// TIA Portal V15.1 export
// export: Created 2024-06-21T08:41:00.9803831Z, ExportSetting WithDefaults, DisplayName Totally Integrated Automation Portal, DisplayVersion V15.1 Update 5, DisplayName TIA Portal Openness, DisplayVersion V15.1 Update 5, DisplayName SINAMICS Startdrive Advanced, DisplayVersion V15.1, DisplayName G130, G150, S120, S150, SINAMICS MV, S210, DisplayVersion V15.1, DisplayName G110M, G120, G120C, G120D, G120P, DisplayVersion V15.1, DisplayName STEP 7 Professional, DisplayVersion V15.1 Update 5, DisplayName STEP 7 Safety, DisplayVersion V15.1, DisplayName WinCC Professional, DisplayVersion V15.1 Update 5, DisplayName SIMATIC Visualization Architect, DisplayVersion V15.1
FUNCTION_BLOCK "LMode"   // FB1000, FBD
TITLE = LMode
{ S7_Optimized_Access := 'FALSE' }
AUTHOR : VCC
FAMILY : Control
NAME : Mode
VERSION : 1.0
// ================================================================================
// This module is used to handle all operating modes for a modezone as well as 
// resetting of alarms. It get the input from LModeSelector.
// ================================================================================
// stored: AutoNumber false, IsIECCheckEnabled false, SetENOAutomatically False, UDAEnableTagReadback false
   VAR_INPUT
      I_NormalStop { ExternalAccessible := 'False'; ExternalVisible := 'False'; ExternalWritable := 'False'} : Bool;   // Normal Stop Activated Stop Automatic
      I_EnableAlarms { ExternalAccessible := 'False'; ExternalVisible := 'False'; ExternalWritable := 'False'} : Bool;   // Filter alarms for lower levels
      I_AutoModeSel { ExternalAccessible := 'False'; ExternalVisible := 'False'; ExternalWritable := 'False'} : Bool;   // Auto selected
      I_StepModeSel { ExternalAccessible := 'False'; ExternalVisible := 'False'; ExternalWritable := 'False'} : Bool;   // Step selected
      I_HomeRunModeSel { ExternalAccessible := 'False'; ExternalVisible := 'False'; ExternalWritable := 'False'} : Bool;   // Homerun selected
      I_HomeRunPush { ExternalAccessible := 'False'; ExternalVisible := 'False'; ExternalWritable := 'False'} : Bool;   // The reset button needs to be active during the homerun
      I_ManualModeSel { ExternalAccessible := 'False'; ExternalVisible := 'False'; ExternalWritable := 'False'} : Bool;   // Manual selected
      I_ForcedManActSel { ExternalAccessible := 'False'; ExternalVisible := 'False'; ExternalWritable := 'False'} : Bool;   // Forced manual key switch
      I_HomerunCond { ExternalAccessible := 'False'; ExternalVisible := 'False'; ExternalWritable := 'False'} : Bool;   // Condition for homerun
      I_HomePos { ExternalAccessible := 'False'; ExternalVisible := 'False'; ExternalWritable := 'False'} : Bool;   // Station in homposition
      I_AfterHomerunSel { ExternalAccessible := 'False'; ExternalVisible := 'False'; ExternalWritable := 'False'} : Bool;   // Show selection after Homrun on HMI
      I_HomeRunRedoSel { ExternalAccessible := 'False'; ExternalVisible := 'False'; ExternalWritable := 'False'} : Bool;   // Redo after Homerun selected
      I_HomeRunWorkDoneSel { ExternalAccessible := 'False'; ExternalVisible := 'False'; ExternalWritable := 'False'} : Bool;   // WorkDone after Homerun selected
      I_HomeRunRedoReset { ExternalAccessible := 'False'; ExternalVisible := 'False'; ExternalWritable := 'False'} : Bool;   // Reset redo after homerun
      I_HomeRunWorkDoneReset { ExternalAccessible := 'False'; ExternalVisible := 'False'; ExternalWritable := 'False'} : Bool;   // Reset workdone after homerun
      I_HomeRunPriorityRedo { ExternalAccessible := 'False'; ExternalVisible := 'False'; ExternalWritable := 'False'} : Bool;   // Priority Redo after homerun
      I_CycleFinishedSel { ExternalAccessible := 'False'; ExternalVisible := 'False'; ExternalWritable := 'False'} : Bool;   // Cycle finished is selected
      I_StartPBSel { ExternalAccessible := 'False'; ExternalVisible := 'False'; ExternalWritable := 'False'} : Bool;   // Summary of Start buttons
      I_AlarmResetPBSel { ExternalAccessible := 'False'; ExternalVisible := 'False'; ExternalWritable := 'False'} : Bool;   // Summary of Alarm reset buttons
      I_PBSetSel { ExternalAccessible := 'False'; ExternalVisible := 'False'; ExternalWritable := 'False'} : Bool;   // Pushbutton Set
      I_PBResetSel { ExternalAccessible := 'False'; ExternalVisible := 'False'; ExternalWritable := 'False'} : Bool;   // Pushbutton Reset
      I_ResetSeqSel { ExternalAccessible := 'False'; ExternalVisible := 'False'; ExternalWritable := 'False'} : Bool;   // Reset Sequence
      I_ResetTMSel { ExternalAccessible := 'False'; ExternalVisible := 'False'; ExternalWritable := 'False'} : Bool;   // Reset Transport memory
      I_SafetyOk { ExternalAccessible := 'False'; ExternalVisible := 'False'; ExternalWritable := 'False'} : Bool;   // SafetyOk / No Haltbutton is activate
      I_NotHaltButton { ExternalAccessible := 'False'; ExternalVisible := 'False'; ExternalWritable := 'False'} : Bool;   // No Haltbutton is activate
      I_ExtAutoCond { ExternalAccessible := 'False'; ExternalVisible := 'False'; ExternalWritable := 'False'} : Bool;   // External Auto Conditions / No Haltbutton is activate
      I_AlarmABCondition { ExternalAccessible := 'False'; ExternalVisible := 'False'; ExternalWritable := 'False'} : Bool;   // Alarm AB condition in the Modezone / Alarm AB condition
      I_AlarmA { ExternalAccessible := 'False'; ExternalVisible := 'False'; ExternalWritable := 'False'} : Bool;   // Alarm A active in the Modezone / Alarm A active in the modezone
      I_AlarmB { ExternalAccessible := 'False'; ExternalVisible := 'False'; ExternalWritable := 'False'} : Bool;   // Alarm B active in the Modezone / Alarm B active in the modezone
      I_AlarmC { ExternalAccessible := 'False'; ExternalVisible := 'False'; ExternalWritable := 'False'} : Bool;   // Alarm C active in the Modezone / Alarm C active in the modezone
      I_AlarmD { ExternalAccessible := 'False'; ExternalVisible := 'False'; ExternalWritable := 'False'} : Bool;   // Alarm D active in the Modezone
      I_UpperLevelZSAlarmABCondition { ExternalAccessible := 'False'; ExternalVisible := 'False'; ExternalWritable := 'False'} : Bool;   // Alarm AB condition from the Safety Zone / Alarm AB condition
      I_UpperLevelZSAlarmA { ExternalAccessible := 'False'; ExternalVisible := 'False'; ExternalWritable := 'False'} : Bool;   // Alarm A active from the Safety Zone / Alarm A active from the top level
      I_UpperLevelZSAlarmB { ExternalAccessible := 'False'; ExternalVisible := 'False'; ExternalWritable := 'False'} : Bool;   // Alarm B active from the Safety Zone / Alarm B active from the top level
      I_UpperLevelZSAlarmC { ExternalAccessible := 'False'; ExternalVisible := 'False'; ExternalWritable := 'False'} : Bool;   // Alarm C active from the Safety Zone / Alarm C active from the top level
      I_UpperLevelZSAlarmD { ExternalAccessible := 'False'; ExternalVisible := 'False'; ExternalWritable := 'False'} : Bool;   // Alarm D active from the Safety Zone
      I_UpperLevelPLCAlarmABCondition { ExternalAccessible := 'False'; ExternalVisible := 'False'; ExternalWritable := 'False'} : Bool;   // Alarm AB condition from the PLC level / Alarm AB condition
      I_UpperLevelPLCAlarmA { ExternalAccessible := 'False'; ExternalVisible := 'False'; ExternalWritable := 'False'} : Bool;   // Alarm A active from the PLC level / Alarm A active from the top level
      I_UpperLevelPLCAlarmB { ExternalAccessible := 'False'; ExternalVisible := 'False'; ExternalWritable := 'False'} : Bool;   // Alarm B active from the PLC level / Alarm B active from the top level
      I_UpperLevelPLCAlarmC { ExternalAccessible := 'False'; ExternalVisible := 'False'; ExternalWritable := 'False'} : Bool;   // Alarm C active from the PLC level / Alarm C active from the top level
      I_UpperLevelPLCAlarmD { ExternalAccessible := 'False'; ExternalVisible := 'False'; ExternalWritable := 'False'} : Bool;   // Alarm D active from the PLC level
      I_AutoModeWarningTime { ExternalAccessible := 'False'; ExternalVisible := 'False'; ExternalWritable := 'False'} : Int;   // Auto Mode warning time / Auto mode warning time
   END_VAR
   VAR_OUTPUT
      O_AutoMode { ExternalAccessible := 'False'; ExternalVisible := 'False'; ExternalWritable := 'False'} : Bool;   // Auto Mode / Auto mode
      O_StepMode { ExternalAccessible := 'False'; ExternalVisible := 'False'; ExternalWritable := 'False'} : Bool;   // Step Mode / Step mode
      O_HomeRunMode { ExternalAccessible := 'False'; ExternalVisible := 'False'; ExternalWritable := 'False'} : Bool;   // Homrun Mode / Homrun mode
      O_ManualMode { ExternalAccessible := 'False'; ExternalVisible := 'False'; ExternalWritable := 'False'} : Bool;   // Manual Mode / Manual mode
      O_ForcedMan { ExternalAccessible := 'False'; ExternalVisible := 'False'; ExternalWritable := 'False'} : Bool;   // Forced manual
      O_AutoStepRun { ExternalAccessible := 'False'; ExternalVisible := 'False'; ExternalWritable := 'False'} : Bool;   // Auto Mode or Step Mode and StartPB is active / Auto mode or Step mode and StartPB is active
      O_AutoStepHomeRunAct { ExternalAccessible := 'False'; ExternalVisible := 'False'; ExternalWritable := 'False'} : Bool;   // Auto, Step or Homerun Mode is active / Auto, Step or Homerun mode is active
      O_StartPB { ExternalAccessible := 'False'; ExternalVisible := 'False'; ExternalWritable := 'False'} : Bool;   // Start button is activated
      O_AlarmResetPB { ExternalAccessible := 'False'; ExternalVisible := 'False'; ExternalWritable := 'False'} : Bool;   // Alarm reset button is activated
      O_SetPBMan { ExternalAccessible := 'False'; ExternalVisible := 'False'; ExternalWritable := 'False'} : Bool;   // Set pushbutton is activated in manual
      O_ResetPBMan { ExternalAccessible := 'False'; ExternalVisible := 'False'; ExternalWritable := 'False'} : Bool;   // Reset pushbutton is activated in manual
      O_ResetTM { ExternalAccessible := 'False'; ExternalVisible := 'False'; ExternalWritable := 'False'} : Bool;   // Reset transport memory
      O_ResetSeq { ExternalAccessible := 'False'; ExternalVisible := 'False'; ExternalWritable := 'False'} : Bool;   // Reset sequence
      O_CycleFinished { ExternalAccessible := 'False'; ExternalVisible := 'False'; ExternalWritable := 'False'} : Bool;   // Cycle finished
      O_AlarmABAct { ExternalAccessible := 'False'; ExternalVisible := 'False'; ExternalWritable := 'False'} : Bool;   // A or B alarm active
      O_HaltButton { ExternalAccessible := 'False'; ExternalVisible := 'False'; ExternalWritable := 'False'} : Bool;   // A Haltbutton is activated
      O_AutoModeWarning { ExternalAccessible := 'False'; ExternalVisible := 'False'; ExternalWritable := 'False'} : Bool;   // Auto Mode warning / Auto mode warning
      O_HomeRunRedo { ExternalAccessible := 'False'; ExternalVisible := 'False'; ExternalWritable := 'False'} : Bool;   // Redo work after homerun
      O_HomeRunWorkDone { ExternalAccessible := 'False'; ExternalVisible := 'False'; ExternalWritable := 'False'} : Bool;   // WorkDone after homerun
      O_HMIResetPBRedColor { ExternalAccessible := 'False'; ExternalVisible := 'False'; ExternalWritable := 'False'} : Bool;   // Red background color for the Reset button on the HMI
      O_ActiveMode : Word;   // Active Mode / Active mode
      O_SelectedMode : Word;   // Selected Mode. Only active when a Mode is selected but not started / Selected mode. Only active when a mode is selected but not started
      O_AlarmABCondition { ExternalAccessible := 'False'; ExternalVisible := 'False'; ExternalWritable := 'False'} : Bool;   // Alarm AB condition
      O_AlarmA { ExternalAccessible := 'False'; ExternalVisible := 'False'; ExternalWritable := 'False'} : Bool;   // Alarms A
      O_AlarmB { ExternalAccessible := 'False'; ExternalVisible := 'False'; ExternalWritable := 'False'} : Bool;   // Alarms B
      O_AlarmC { ExternalAccessible := 'False'; ExternalVisible := 'False'; ExternalWritable := 'False'} : Bool;   // Alarms C
      O_AlarmD { ExternalAccessible := 'False'; ExternalVisible := 'False'; ExternalWritable := 'False'} : Bool;   // Alarms D
      H_AlarmWord { ExternalAccessible := 'False'; ExternalVisible := 'False'; ExternalWritable := 'False'} : DWord;   // Alarm Word
   END_VAR
   VAR_IN_OUT
      IO_Modes : "Modes";
   END_VAR
   VAR DB_SPECIFIC
      AC_HomeRun { ExternalAccessible := 'False'; ExternalVisible := 'False'; ExternalWritable := 'False'} : Bool;   // Homerun alarm
      AC_AutoNotStarted { ExternalAccessible := 'False'; ExternalVisible := 'False'; ExternalWritable := 'False'} : Bool;   // Auto not started
      AC_StartPBSticking { ExternalAccessible := 'False'; ExternalVisible := 'False'; ExternalWritable := 'False'} : Bool;   // Start push button is ON longer then 20 sec
      AC_ResetPBSticking { ExternalAccessible := 'False'; ExternalVisible := 'False'; ExternalWritable := 'False'} : Bool;   // Reset Alarm push button is ON longer then 20 sec
      AD_ManualMode { ExternalAccessible := 'False'; ExternalVisible := 'False'; ExternalWritable := 'False'} : Bool;   // Manual Mode activated / Manual mode activated
      AD_StepModeSel { ExternalAccessible := 'False'; ExternalVisible := 'False'; ExternalWritable := 'False'} : Bool;   // Step Mode selected / Step mode selected
      AD_HomeRunMode { ExternalAccessible := 'False'; ExternalVisible := 'False'; ExternalWritable := 'False'} : Bool;   // Homerun Mode activated / Homerun mode activated
      AE_NormalStop { ExternalAccessible := 'False'; ExternalVisible := 'False'; ExternalWritable := 'False'} : Bool;   // Normal Stop Mode Activated / Normal Stop Mode activated / NormalStop Aktiverat
      AE_ResetSeq { ExternalAccessible := 'False'; ExternalVisible := 'False'; ExternalWritable := 'False'} : Bool;   // Reset sequence activated
      AE_ResetTM { ExternalAccessible := 'False'; ExternalVisible := 'False'; ExternalWritable := 'False'} : Bool;   // Reset Transport memory activated
      AE_ForcedMan { ExternalAccessible := 'False'; ExternalVisible := 'False'; ExternalWritable := 'False'} : Bool;   // Manual Forced activated
      H_Anim : Word;   // Animation
      H_Anim2 : Word;   // Animation
      H_HomeRunModeAnim : Word;   // Homerun Animation
      H_ConfigBtnResetTM : Bool;   // From the HMI - Config internal tag
      H_ConfigBtnResetSeq : Bool;   // From the HMI - Config internal tag
      H_ModeChanged : Bool;   // From the HMI - Mode changed to Auto
      H_ScreenChanged : Bool;   // From the HMI - The screen has changed
      HomeRunHold { ExternalAccessible := 'False'; ExternalVisible := 'False'; ExternalWritable := 'False'} : Bool;   // Homerun, the operator have to hold the button
      HomeRunMc { ExternalAccessible := 'False'; ExternalVisible := 'False'; ExternalWritable := 'False'} : Bool;   // Homerun without hold function
      AlarmA { ExternalAccessible := 'False'; ExternalVisible := 'False'; ExternalWritable := 'False'} : Bool;   // Alarm A active in the FB
      AlarmB { ExternalAccessible := 'False'; ExternalVisible := 'False'; ExternalWritable := 'False'} : Bool;   // Alarm B active in the FB
      AlarmC { ExternalAccessible := 'False'; ExternalVisible := 'False'; ExternalWritable := 'False'} : Bool;   // Alarm C active in the FB
      AlarmD { ExternalAccessible := 'False'; ExternalVisible := 'False'; ExternalWritable := 'False'} : Bool;   // Alarm D active in the FB
      StepPulse { ExternalAccessible := 'False'; ExternalVisible := 'False'; ExternalWritable := 'False'} : Bool;   // Step pulse
      AutoMode { ExternalAccessible := 'False'; ExternalVisible := 'False'; ExternalWritable := 'False'} : Bool;   // Auto Mode / Auto mode
      StepMode { ExternalAccessible := 'False'; ExternalVisible := 'False'; ExternalWritable := 'False'} : Bool;   // Step Mode / Step mode
      HomeRunMode { ExternalAccessible := 'False'; ExternalVisible := 'False'; ExternalWritable := 'False'} : Bool;   // Homrun Mode / Homrun mode
      ManualMode { ExternalAccessible := 'False'; ExternalVisible := 'False'; ExternalWritable := 'False'} : Bool;   // Manual Mode / Manual mode
      ForcedMan { ExternalAccessible := 'False'; ExternalVisible := 'False'; ExternalWritable := 'False'} : Bool;   // Forced manual
      AutoStepRun { ExternalAccessible := 'False'; ExternalVisible := 'False'; ExternalWritable := 'False'} : Bool;   // Auto Mode or Step Mode and StartPB is active / Auto mode or Step mode and StartPB is active
      AutoStepHomeRunAct { ExternalAccessible := 'False'; ExternalVisible := 'False'; ExternalWritable := 'False'} : Bool;   // Auto, Step or Homerun Mode is active / Auto, Step or Homerun mode is active
      SetPBMan { ExternalAccessible := 'False'; ExternalVisible := 'False'; ExternalWritable := 'False'} : Bool;   // Set pushbutton is activated in manual
      ResetPBMan { ExternalAccessible := 'False'; ExternalVisible := 'False'; ExternalWritable := 'False'} : Bool;   // Reset pushbutton is activated in manual
      ResetTM { ExternalAccessible := 'False'; ExternalVisible := 'False'; ExternalWritable := 'False'} : Bool;   // Reset transport memory
      ResetSeq { ExternalAccessible := 'False'; ExternalVisible := 'False'; ExternalWritable := 'False'} : Bool;   // Reset sequence
      HomeRunAlmCond { ExternalAccessible := 'False'; ExternalVisible := 'False'; ExternalWritable := 'False'} : Bool;   // Homerun alarm condition
      HomeRunRedo { ExternalAccessible := 'False'; ExternalVisible := 'False'; ExternalWritable := 'False'} : Bool;   // Redo work after homerun
      HomeRunWorkDone { ExternalAccessible := 'False'; ExternalVisible := 'False'; ExternalWritable := 'False'} : Bool;   // WorkDone after homerun
      HomeRunModeNegEdge1 { ExternalAccessible := 'False'; ExternalVisible := 'False'; ExternalWritable := 'False'} : Bool;   // Negative edge of homerun active
      HomeRunModeNegEdge2 { ExternalAccessible := 'False'; ExternalVisible := 'False'; ExternalWritable := 'False'} : Bool;   // Negative edge of homerun active
      HomeRunModePosEdge1 { ExternalAccessible := 'False'; ExternalVisible := 'False'; ExternalWritable := 'False'} : Bool;   // Positive edge of homerun active
      HomeRunModePosEdge2 { ExternalAccessible := 'False'; ExternalVisible := 'False'; ExternalWritable := 'False'} : Bool;   // Positive edge of homerun active
      AutoModeWarningTimer { ExternalAccessible := 'False'; ExternalVisible := 'False'; ExternalWritable := 'False'} : Bool;   // Auto Mode warning timer / Auto mode warning timer
      TimerResetSeq { ExternalAccessible := 'False'; ExternalVisible := 'False'; ExternalWritable := 'False'} : Bool;   // Timer for reset sequence
      TimerResetTM { ExternalAccessible := 'False'; ExternalVisible := 'False'; ExternalWritable := 'False'} : Bool;   // Timer for reset TM
      AutoModeWarning { ExternalAccessible := 'False'; ExternalVisible := 'False'; ExternalWritable := 'False'} : Bool;   // Auto Mode warning / Auto mode warning
      AutoModeWarningRunning { ExternalAccessible := 'False'; ExternalVisible := 'False'; ExternalWritable := 'False'} : DInt;   // Auto Mode warning timmer running / Auto mode warning timmer running
      StartAutoWarning { ExternalAccessible := 'False'; ExternalVisible := 'False'; ExternalWritable := 'False'} : Bool;   // Start button Auto warning
      StartPBSel { ExternalAccessible := 'False'; ExternalVisible := 'False'; ExternalWritable := 'False'} : Bool;   // Summary of Start buttons
      AlarmResetPBSel { ExternalAccessible := 'False'; ExternalVisible := 'False'; ExternalWritable := 'False'} : Bool;   // Summary of Alarm reset buttons
   END_VAR
   VAR
      TimerAutoWarning { ExternalAccessible := 'False'; ExternalVisible := 'False'; ExternalWritable := 'False'} : "LTimer";   // Timer
      TimerResetSequence { ExternalAccessible := 'False'; ExternalVisible := 'False'; ExternalWritable := 'False'} : "LTimer";   // Timer
      TimerAutoNotStarted { ExternalAccessible := 'False'; ExternalVisible := 'False'; ExternalWritable := 'False'} : "LTimer";   // Timer
      TimerStartBtnStuck { ExternalAccessible := 'False'; ExternalVisible := 'False'; ExternalWritable := 'False'} : "LTimer";   // Timer to maximize the pulse on the Start PB
      TimerResetBtnStuck { ExternalAccessible := 'False'; ExternalVisible := 'False'; ExternalWritable := 'False'} : "LTimer";   // Timer to maximize the pulse on the Reset PB
      TimerResetTransportMem { ExternalAccessible := 'False'; ExternalVisible := 'False'; ExternalWritable := 'False'} : "LTimer";   // Timer to extend Reset TM
   END_VAR
   VAR DB_SPECIFIC
      TimerStartPBSel { ExternalAccessible := 'False'; ExternalVisible := 'False'; ExternalWritable := 'False'} : TOF_TIME;   // Timer
      TimerAlarmResetPBSel { ExternalAccessible := 'False'; ExternalVisible := 'False'; ExternalWritable := 'False'} : TOF_TIME;   // Timer
      TimerModeChanged { ExternalAccessible := 'False'; ExternalVisible := 'False'; ExternalWritable := 'False'} : TON_TIME;   // Timer
      TimerScreenChanged { ExternalAccessible := 'False'; ExternalVisible := 'False'; ExternalWritable := 'False'} : TON_TIME;   // Timer
   END_VAR
   VAR_TEMP
      AutoModeWarnMillieSec : DInt;   // Auto Mode warning millie seconds / Auto mode warning millie seconds
      AutoModeWarnSec : DInt;   // Auto Mode warning seconds / Auto mode warning seconds
      AlarmABConditionActive : Bool;   // Alarm AB condition Active in the Modezone / Alarm AB condition
      AlarmAActive : Bool;   // Alarm A Active in the Modezone
      AlarmBActive : Bool;   // Alarm B Active in the Modezone
      AlarmCActive : Bool;   // Alarm C Active in the Modezone
      AlarmDActive : Bool;   // Alarm D Active in the Modezone
   END_VAR
   VAR_TEMP   // added for the SCL form of the ladder/FBD networks
      _w1 : Bool;
      _w2 : Bool;
   END_VAR
BEGIN

REGION Network 1: **** 1 - Inputs **** The Mode has changed
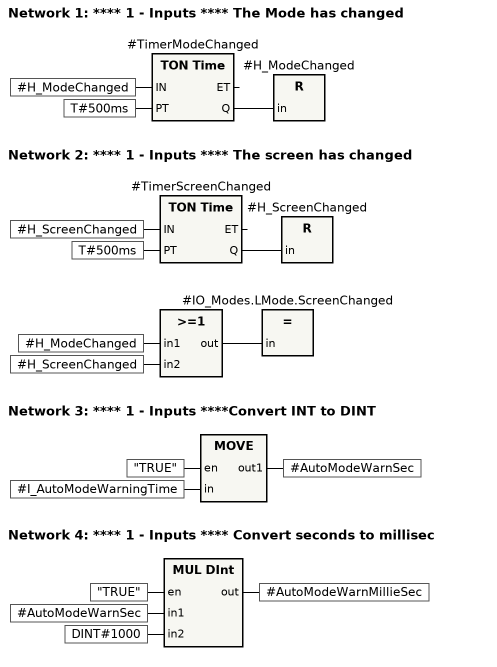
   #TimerModeChanged(IN := #H_ModeChanged, PT := T#500ms);   // TON
   IF #TimerModeChanged.Q THEN #H_ModeChanged := FALSE; END_IF;
END_REGION

REGION Network 2: **** 1 - Inputs **** The screen has changed
   #TimerScreenChanged(IN := #H_ScreenChanged, PT := T#500ms);   // TON
   IF #TimerScreenChanged.Q THEN #H_ScreenChanged := FALSE; END_IF;
   #IO_Modes.LMode.ScreenChanged := #H_ModeChanged OR #H_ScreenChanged;
END_REGION

REGION Network 3: **** 1 - Inputs ****Convert INT to DINT
   // Convert INT to DINT
   IF "TRUE" THEN #AutoModeWarnSec := #I_AutoModeWarningTime; END_IF;
END_REGION

REGION Network 4: **** 1 - Inputs **** Convert seconds to millisec
   // Convert seconds to millisec
   IF "TRUE" THEN #AutoModeWarnMillieSec := #AutoModeWarnSec * DINT#1000; END_IF;
END_REGION

REGION Network 5: **** 1 - Inputs **** Alarms Upperlevel And ModeZone Objects
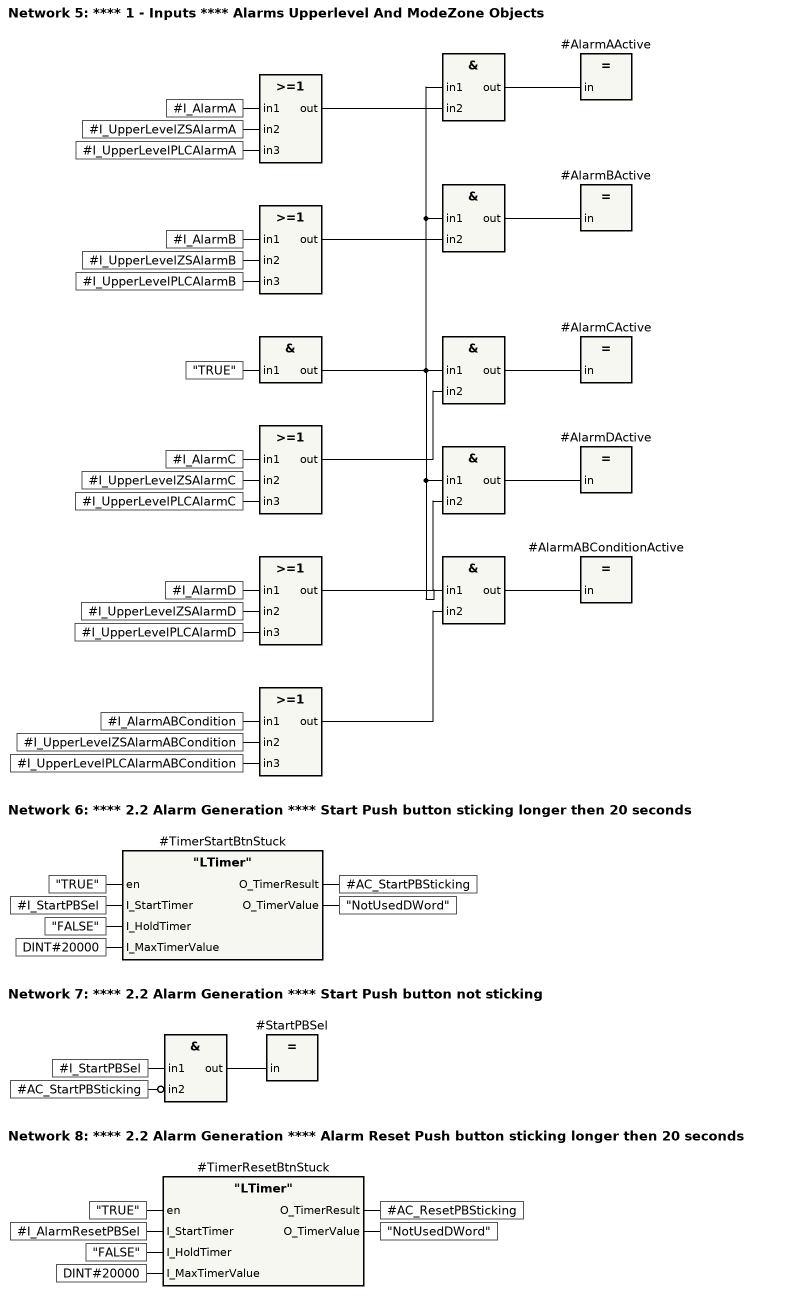
   #AlarmAActive := "TRUE" AND (#I_AlarmA OR #I_UpperLevelZSAlarmA OR #I_UpperLevelPLCAlarmA);
   #AlarmBActive := "TRUE" AND (#I_AlarmB OR #I_UpperLevelZSAlarmB OR #I_UpperLevelPLCAlarmB);
   #AlarmCActive := "TRUE" AND (#I_AlarmC OR #I_UpperLevelZSAlarmC OR #I_UpperLevelPLCAlarmC);
   #AlarmDActive := "TRUE" AND (#I_AlarmD OR #I_UpperLevelZSAlarmD OR #I_UpperLevelPLCAlarmD);
   #AlarmABConditionActive := "TRUE" AND (#I_AlarmABCondition OR #I_UpperLevelZSAlarmABCondition OR #I_UpperLevelPLCAlarmABCondition);
END_REGION

REGION Network 6: **** 2.2 Alarm Generation **** Start Push button sticking longer then 20 seconds
   // Start Push button sticking longer then 20 seconds
   IF "TRUE" THEN
       #TimerStartBtnStuck(I_StartTimer := #I_StartPBSel,   // "LTimer"
                           I_HoldTimer := "FALSE",
                           I_MaxTimerValue := DINT#20000,
                           O_TimerResult => #AC_StartPBSticking,
                           O_TimerValue => "NotUsedDWord");
   END_IF;
END_REGION

REGION Network 7: **** 2.2 Alarm Generation **** Start Push button not sticking
   // Start Push button not sticking
   #StartPBSel := #I_StartPBSel AND NOT #AC_StartPBSticking;
END_REGION

REGION Network 8: **** 2.2 Alarm Generation **** Alarm Reset Push button sticking longer then 20 seconds
   // Alarm Reset Push button sticking longer then 20 seconds
   IF "TRUE" THEN
       #TimerResetBtnStuck(I_StartTimer := #I_AlarmResetPBSel,   // "LTimer"
                           I_HoldTimer := "FALSE",
                           I_MaxTimerValue := DINT#20000,
                           O_TimerResult => #AC_ResetPBSticking,
                           O_TimerValue => "NotUsedDWord");
   END_IF;
END_REGION

REGION Network 9: **** 2.2 Alarm Generation **** Alarm Reset Push button not sticking
   // Alarm Reset Push button not sticking
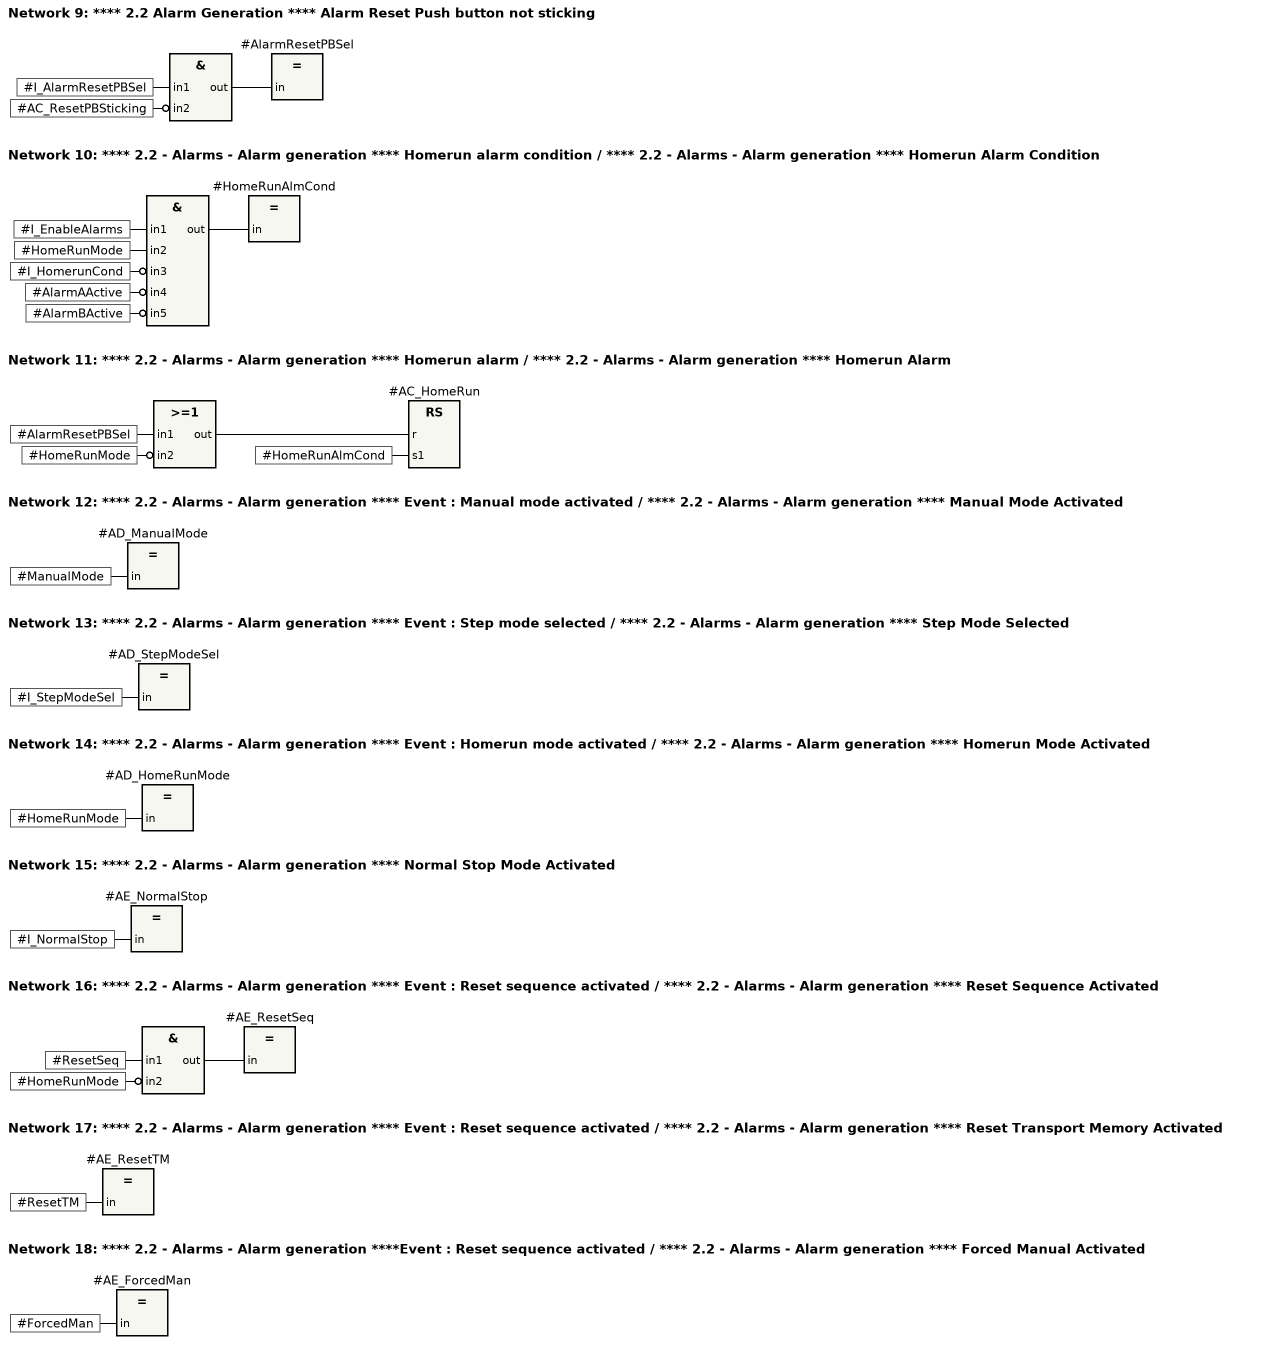
   #AlarmResetPBSel := #I_AlarmResetPBSel AND NOT #AC_ResetPBSticking;
END_REGION

REGION Network 10: **** 2.2 - Alarms - Alarm generation **** Homerun alarm condition / **** 2.2 - Alarms - Alarm generation **** Homerun Alarm Condition
   // Homerun alarm condition
   #HomeRunAlmCond := #I_EnableAlarms AND #HomeRunMode AND NOT #I_HomerunCond AND NOT #AlarmAActive AND NOT #AlarmBActive;
END_REGION

REGION Network 11: **** 2.2 - Alarms - Alarm generation **** Homerun alarm / **** 2.2 - Alarms - Alarm generation **** Homerun Alarm
   // Homerun alarm
   IF #AlarmResetPBSel OR NOT #HomeRunMode THEN
       #AC_HomeRun := FALSE;   // RS flip-flop
   END_IF;
   IF #HomeRunAlmCond THEN #AC_HomeRun := TRUE; END_IF;
END_REGION

REGION Network 12: **** 2.2 - Alarms - Alarm generation **** Event : Manual mode activated / **** 2.2 - Alarms - Alarm generation **** Manual Mode Activated
   // Event : Manual mode activated / Event : Manual Mode activated
   #AD_ManualMode := #ManualMode;
END_REGION

REGION Network 13: **** 2.2 - Alarms - Alarm generation **** Event : Step mode selected / **** 2.2 - Alarms - Alarm generation **** Step Mode Selected
   // Event : Step mode selected / Event : Step Mode selected
   #AD_StepModeSel := #I_StepModeSel;
END_REGION

REGION Network 14: **** 2.2 - Alarms - Alarm generation **** Event : Homerun mode activated / **** 2.2 - Alarms - Alarm generation **** Homerun Mode Activated
   // Event : Homerun mode activated / Event : Homerun Mode activated
   #AD_HomeRunMode := #HomeRunMode;
END_REGION

REGION Network 15: **** 2.2 - Alarms - Alarm generation **** Normal Stop Mode Activated
   // Event : Normal Stop Mode activated
   #AE_NormalStop := #I_NormalStop;
END_REGION

REGION Network 16: **** 2.2 - Alarms - Alarm generation **** Event : Reset sequence activated / **** 2.2 - Alarms - Alarm generation **** Reset Sequence Activated
   // Event : Reset sequence activated
   #AE_ResetSeq := #ResetSeq AND NOT #HomeRunMode;
END_REGION

REGION Network 17: **** 2.2 - Alarms - Alarm generation **** Event : Reset sequence activated / **** 2.2 - Alarms - Alarm generation **** Reset Transport Memory Activated
   // Event : Reset sequence activated / Event : Reset transport memory activated
   #AE_ResetTM := #ResetTM;
END_REGION

REGION Network 18: **** 2.2 - Alarms - Alarm generation ****Event : Reset sequence activated / **** 2.2 - Alarms - Alarm generation **** Forced Manual Activated
   // Event : Reset sequence activated / Event : Forced manual activated
   #AE_ForcedMan := #ForcedMan;
END_REGION

REGION Network 19: **** 2.2 - Alarms - Alarm generation **** Auto selected, but not started / **** 2.2 - Alarms - Alarm generation **** Auto Selected, But not Started
   // Auto selected, but not started
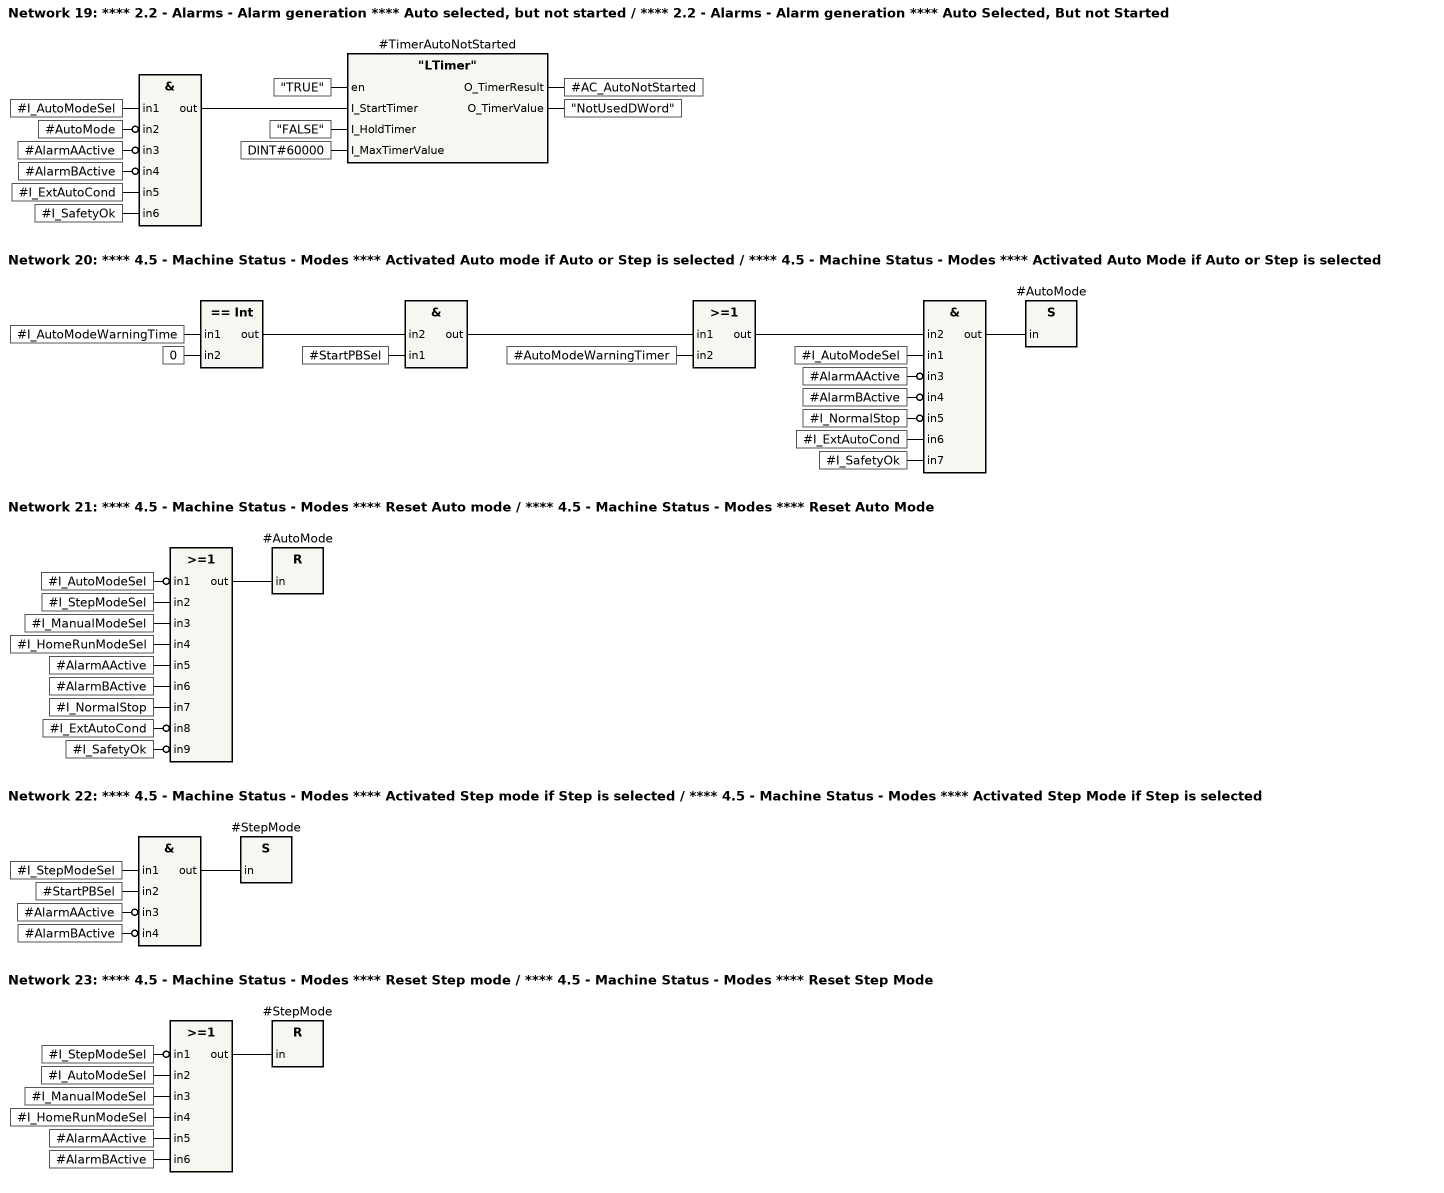
   IF "TRUE" THEN
       #TimerAutoNotStarted(I_StartTimer := #I_AutoModeSel AND NOT #AutoMode AND NOT #AlarmAActive AND NOT #AlarmBActive AND #I_ExtAutoCond AND #I_SafetyOk,   // "LTimer"
                            I_HoldTimer := "FALSE",
                            I_MaxTimerValue := DINT#60000,
                            O_TimerResult => #AC_AutoNotStarted,
                            O_TimerValue => "NotUsedDWord");
   END_IF;
END_REGION

REGION Network 20: **** 4.5 - Machine Status - Modes **** Activated Auto mode if Auto or Step is selected / **** 4.5 - Machine Status - Modes **** Activated Auto Mode if Auto or Step is selected
   // Activated Auto mode if Auto or Step is selected / Activated Auto Mode if Auto or Step is selected
   IF (((#I_AutoModeWarningTime = 0) AND #StartPBSel) OR #AutoModeWarningTimer) AND #I_AutoModeSel AND NOT #AlarmAActive AND NOT #AlarmBActive AND NOT #I_NormalStop AND #I_ExtAutoCond AND #I_SafetyOk THEN
       #AutoMode := TRUE;
   END_IF;
END_REGION

REGION Network 21: **** 4.5 - Machine Status - Modes **** Reset Auto mode / **** 4.5 - Machine Status - Modes **** Reset Auto Mode
   // Reset Auto mode / Reset Auto Mode
   IF NOT #I_AutoModeSel OR #I_StepModeSel OR #I_ManualModeSel OR #I_HomeRunModeSel OR #AlarmAActive OR #AlarmBActive OR #I_NormalStop OR NOT #I_ExtAutoCond OR NOT #I_SafetyOk THEN
       #AutoMode := FALSE;
   END_IF;
END_REGION

REGION Network 22: **** 4.5 - Machine Status - Modes **** Activated Step mode if Step is selected / **** 4.5 - Machine Status - Modes **** Activated Step Mode if Step is selected
   // Activated Step mode if Step is selected / Activated Step Mode if Step is selected
   IF #I_StepModeSel AND #StartPBSel AND NOT #AlarmAActive AND NOT #AlarmBActive THEN
       #StepMode := TRUE;
   END_IF;
END_REGION

REGION Network 23: **** 4.5 - Machine Status - Modes **** Reset Step mode / **** 4.5 - Machine Status - Modes **** Reset Step Mode
   // Reset Step mode / Reset Step Mode
   IF NOT #I_StepModeSel OR #I_AutoModeSel OR #I_ManualModeSel OR #I_HomeRunModeSel OR #AlarmAActive OR #AlarmBActive THEN
       #StepMode := FALSE;
   END_IF;
END_REGION

REGION Network 24: **** 4.5 - Machine Status - Modes **** Activate Homerun mode if all robots are out of station / **** 4.5 - Machine Status - Modes **** Activate Homerun Mode if all robots are out of station
   // Activate Homerun mode if all robots are out of station / Activate Homerun Mode if all robots are out of station
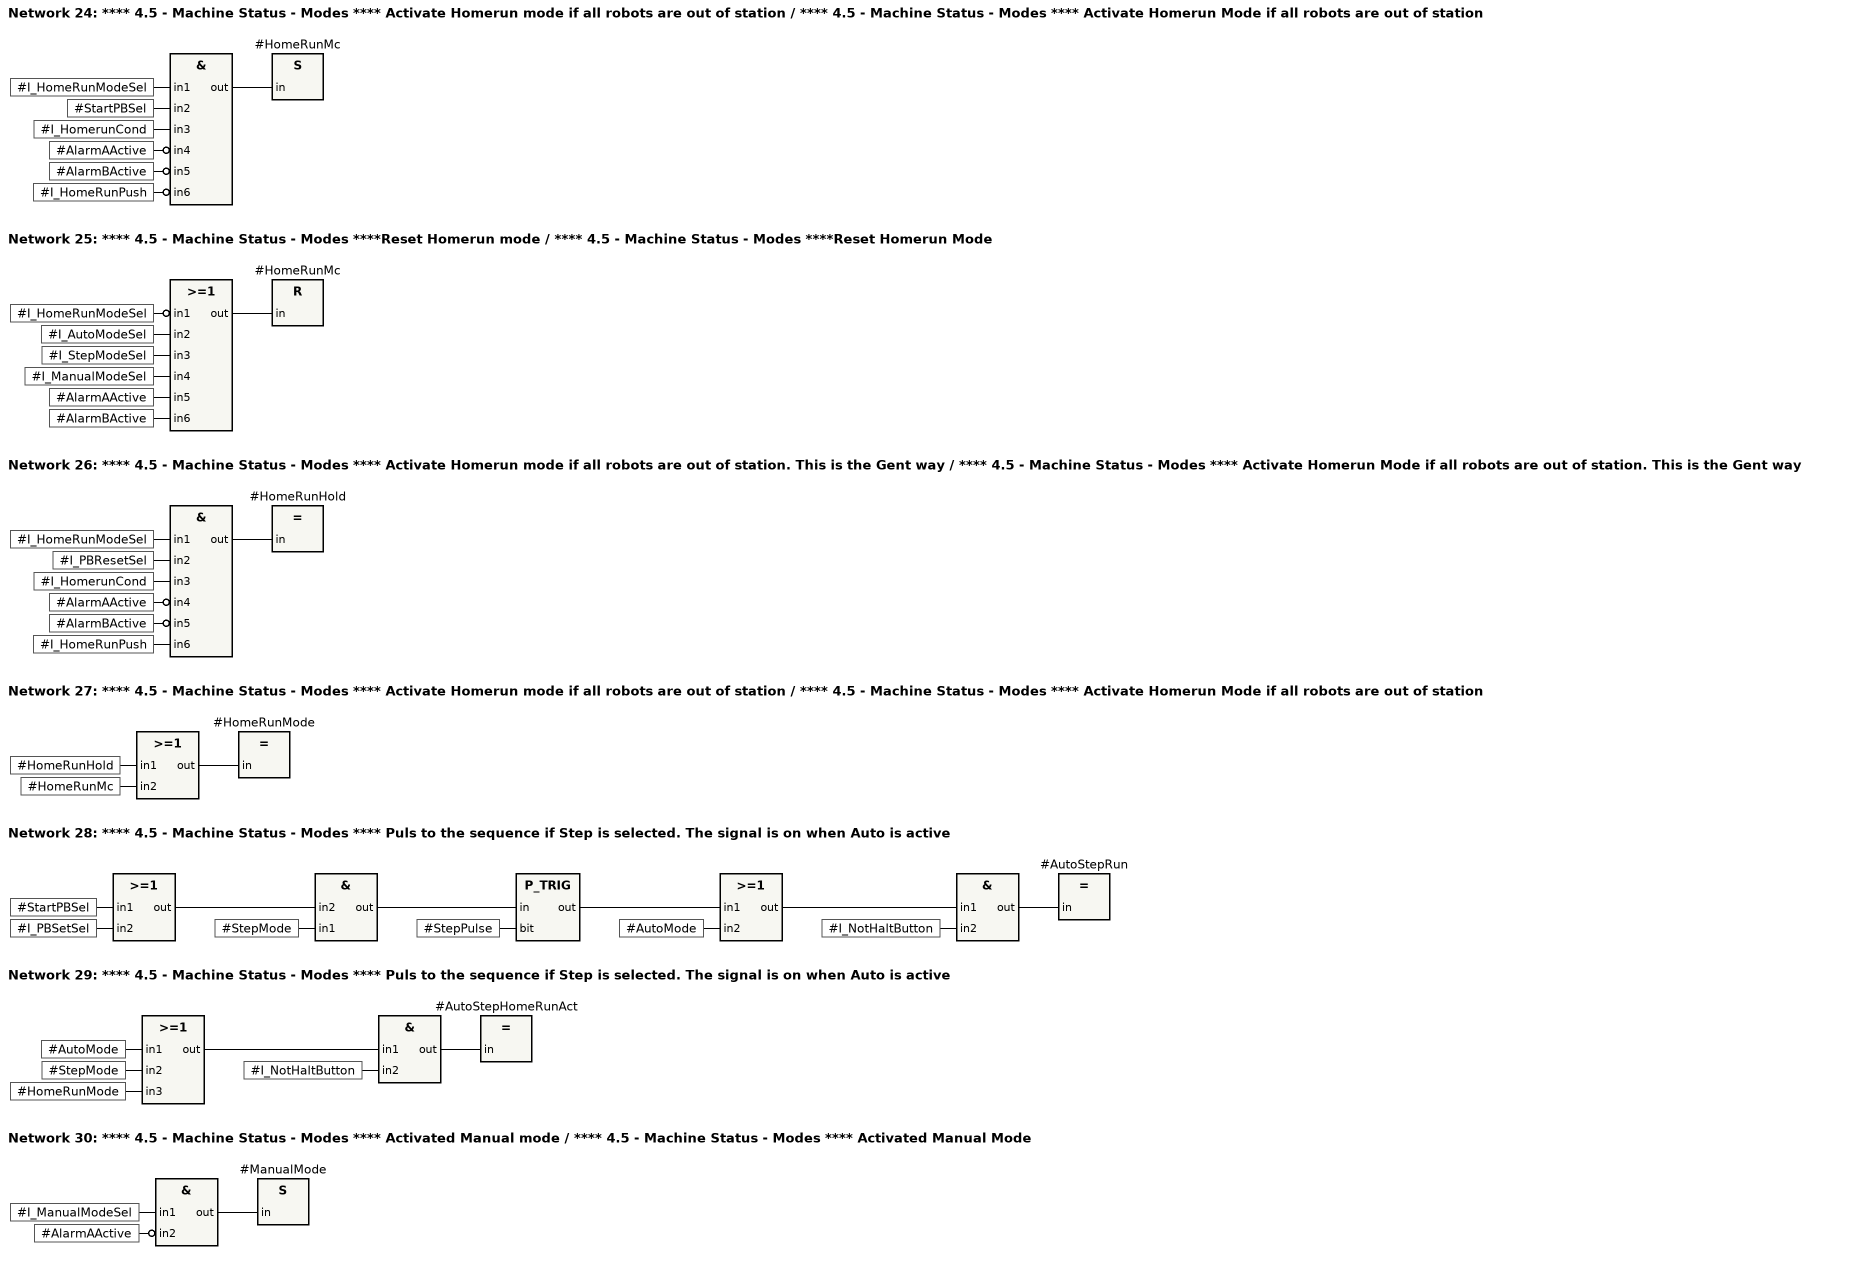
   IF #I_HomeRunModeSel AND #StartPBSel AND #I_HomerunCond AND NOT #AlarmAActive AND NOT #AlarmBActive AND NOT #I_HomeRunPush THEN
       #HomeRunMc := TRUE;
   END_IF;
END_REGION

REGION Network 25: **** 4.5 - Machine Status - Modes ****Reset Homerun mode / **** 4.5 - Machine Status - Modes ****Reset Homerun Mode
   // Reset Homerun mode / Reset Homerun Mode
   IF NOT #I_HomeRunModeSel OR #I_AutoModeSel OR #I_StepModeSel OR #I_ManualModeSel OR #AlarmAActive OR #AlarmBActive THEN
       #HomeRunMc := FALSE;
   END_IF;
END_REGION

REGION Network 26: **** 4.5 - Machine Status - Modes **** Activate Homerun mode if all robots are out of station. This is the Gent way / **** 4.5 - Machine Status - Modes **** Activate Homerun Mode if all robots are out of station. This is the Gent way
   // Activate Homerun mode if all robots are out of station. This is the Gent way 
   // there the reset pushbutton have to be pressed during the complete homerun.
   // Activate Homerun Mode if all robots are out of station. This is the Gent way 
   // there the reset pushbutton have to be pressed during the complete homerun.
   #HomeRunHold := #I_HomeRunModeSel AND #I_PBResetSel AND #I_HomerunCond AND NOT #AlarmAActive AND NOT #AlarmBActive AND #I_HomeRunPush;
END_REGION

REGION Network 27: **** 4.5 - Machine Status - Modes **** Activate Homerun mode if all robots are out of station / **** 4.5 - Machine Status - Modes **** Activate Homerun Mode if all robots are out of station
   // Activate Homerun mode if all robots are out of station. / Activate Homerun Mode if all robots are out of station.
   #HomeRunMode := #HomeRunHold OR #HomeRunMc;
END_REGION

REGION Network 28: **** 4.5 - Machine Status - Modes **** Puls to the sequence if Step is selected. The signal is on when Auto is active
   // Puls to the sequence if Step is selected. The signal is on when Auto is active.
   #_w1 := (#StartPBSel OR #I_PBSetSel) AND #StepMode;
   #_w2 := #_w1 AND NOT #StepPulse;   // rising edge
   #StepPulse := #_w1;
   #AutoStepRun := (#_w2 OR #AutoMode) AND #I_NotHaltButton;
END_REGION

REGION Network 29: **** 4.5 - Machine Status - Modes **** Puls to the sequence if Step is selected. The signal is on when Auto is active
   // Puls to the sequence if Step is selected. The signal is on when Auto is active.
   #AutoStepHomeRunAct := (#AutoMode OR #StepMode OR #HomeRunMode) AND #I_NotHaltButton;
END_REGION

REGION Network 30: **** 4.5 - Machine Status - Modes **** Activated Manual mode / **** 4.5 - Machine Status - Modes **** Activated Manual Mode
   // Activated Manual mode / Activated Manual Mode
   IF #I_ManualModeSel AND NOT #AlarmAActive THEN #ManualMode := TRUE; END_IF;
END_REGION

REGION Network 31: **** 4.5 - Machine Status - Modes **** Reset Manual mode / **** 4.5 - Machine Status - Modes **** Reset Manual Mode
   // Reset Manual mode / Reset Manual Mode
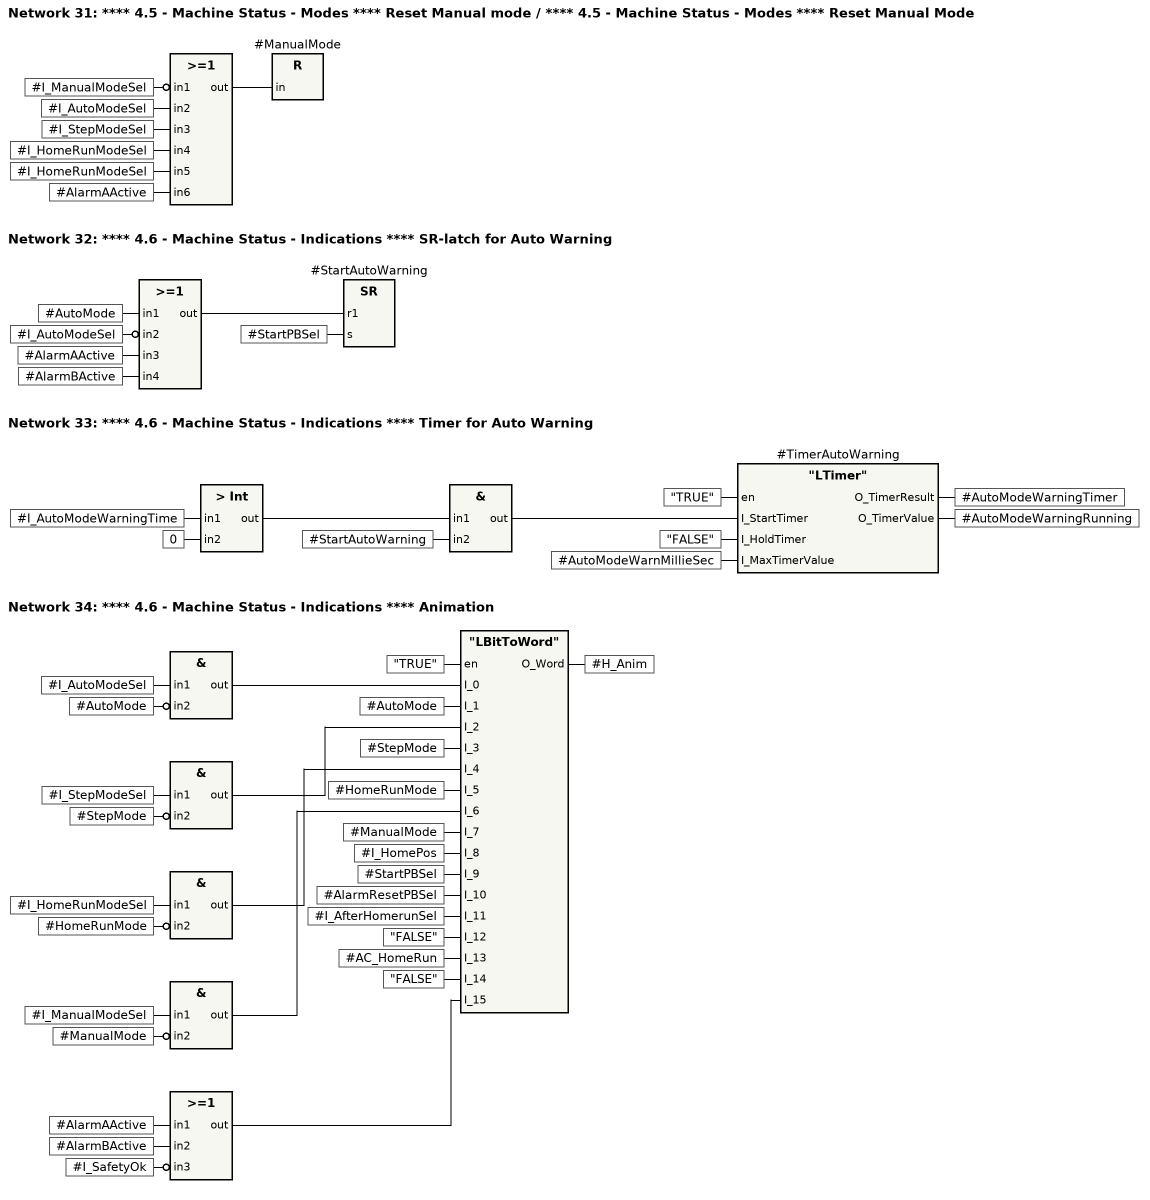
   IF NOT #I_ManualModeSel OR #I_AutoModeSel OR #I_StepModeSel OR #I_HomeRunModeSel OR #I_HomeRunModeSel OR #AlarmAActive THEN
       #ManualMode := FALSE;
   END_IF;
END_REGION

REGION Network 32: **** 4.6 - Machine Status - Indications **** SR-latch for Auto Warning
   // SR-latch for Auto Warning
   IF #StartPBSel THEN
       #StartAutoWarning := TRUE;   // SR flip-flop
   END_IF;
   IF #AutoMode OR NOT #I_AutoModeSel OR #AlarmAActive OR #AlarmBActive THEN
       #StartAutoWarning := FALSE;
   END_IF;
END_REGION

REGION Network 33: **** 4.6 - Machine Status - Indications **** Timer for Auto Warning
   // Timer for Auto Warning
   IF "TRUE" THEN
       #TimerAutoWarning(I_StartTimer := (#I_AutoModeWarningTime > 0) AND #StartAutoWarning,   // "LTimer"
                         I_HoldTimer := "FALSE",
                         I_MaxTimerValue := #AutoModeWarnMillieSec,
                         O_TimerResult => #AutoModeWarningTimer,
                         O_TimerValue => #AutoModeWarningRunning);
   END_IF;
END_REGION

REGION Network 34: **** 4.6 - Machine Status - Indications **** Animation
   // Animation
   IF "TRUE" THEN
       "LBitToWord"(I_0 := #I_AutoModeSel AND NOT #AutoMode,
                    I_1 := #AutoMode,
                    I_2 := #I_StepModeSel AND NOT #StepMode,
                    I_3 := #StepMode,
                    I_4 := #I_HomeRunModeSel AND NOT #HomeRunMode,
                    I_5 := #HomeRunMode,
                    I_6 := #I_ManualModeSel AND NOT #ManualMode,
                    I_7 := #ManualMode,
                    I_8 := #I_HomePos,
                    I_9 := #StartPBSel,
                    I_10 := #AlarmResetPBSel,
                    I_11 := #I_AfterHomerunSel,
                    I_12 := "FALSE",
                    I_13 := #AC_HomeRun,
                    I_14 := "FALSE",
                    I_15 := #AlarmAActive OR #AlarmBActive OR NOT #I_SafetyOk,
                    O_Word => #H_Anim);
   END_IF;
END_REGION

REGION Network 35: **** 4.6 - Machine Status - Indications **** Animation2
   // Animation
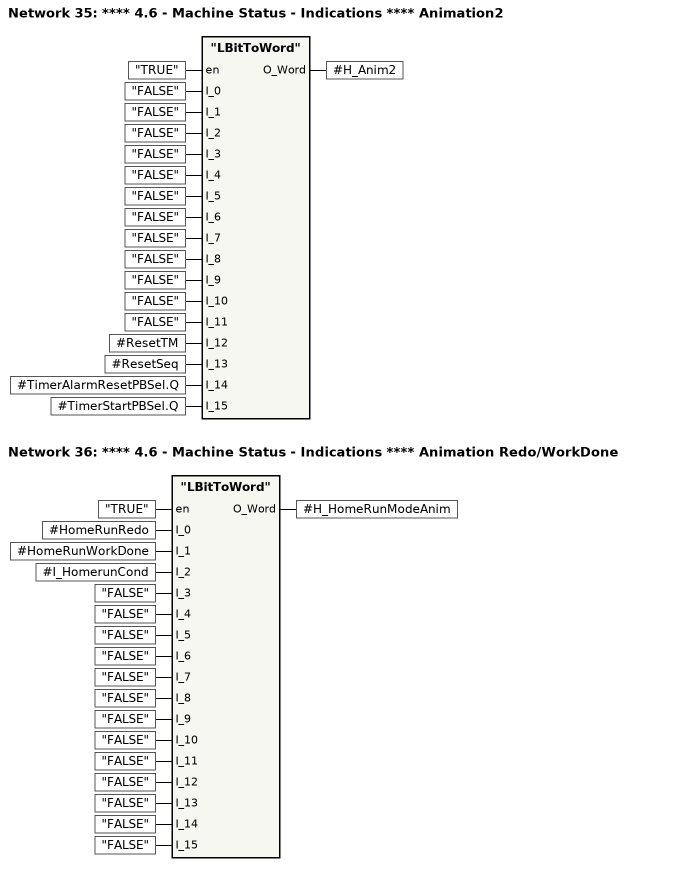
   IF "TRUE" THEN
       "LBitToWord"(I_0 := "FALSE",
                    I_1 := "FALSE",
                    I_2 := "FALSE",
                    I_3 := "FALSE",
                    I_4 := "FALSE",
                    I_5 := "FALSE",
                    I_6 := "FALSE",
                    I_7 := "FALSE",
                    I_8 := "FALSE",
                    I_9 := "FALSE",
                    I_10 := "FALSE",
                    I_11 := "FALSE",
                    I_12 := #ResetTM,
                    I_13 := #ResetSeq,
                    I_14 := #TimerAlarmResetPBSel.Q,
                    I_15 := #TimerStartPBSel.Q,
                    O_Word => #H_Anim2);
   END_IF;
END_REGION

REGION Network 36: **** 4.6 - Machine Status - Indications **** Animation Redo/WorkDone
   // Animation Redo/WorkDone
   IF "TRUE" THEN
       "LBitToWord"(I_0 := #HomeRunRedo,
                    I_1 := #HomeRunWorkDone,
                    I_2 := #I_HomerunCond,
                    I_3 := "FALSE",
                    I_4 := "FALSE",
                    I_5 := "FALSE",
                    I_6 := "FALSE",
                    I_7 := "FALSE",
                    I_8 := "FALSE",
                    I_9 := "FALSE",
                    I_10 := "FALSE",
                    I_11 := "FALSE",
                    I_12 := "FALSE",
                    I_13 := "FALSE",
                    I_14 := "FALSE",
                    I_15 := "FALSE",
                    O_Word => #H_HomeRunModeAnim);
   END_IF;
END_REGION

REGION Network 37: **** 4.6 - Machine Status - Indications **** Animation HMI LED
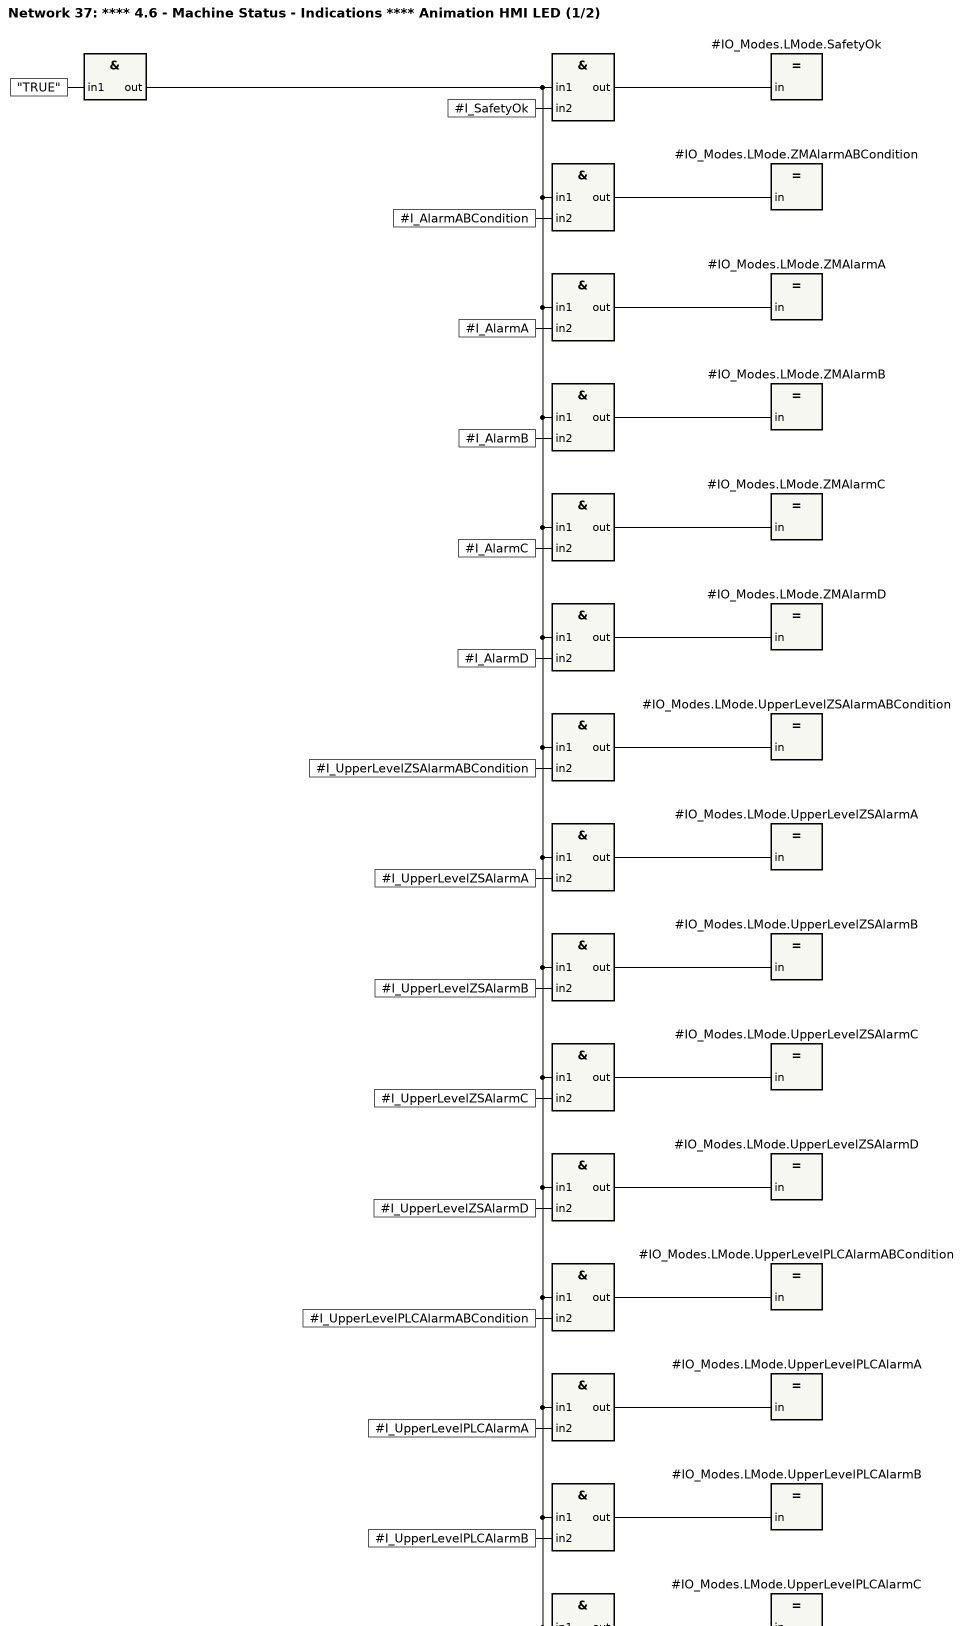
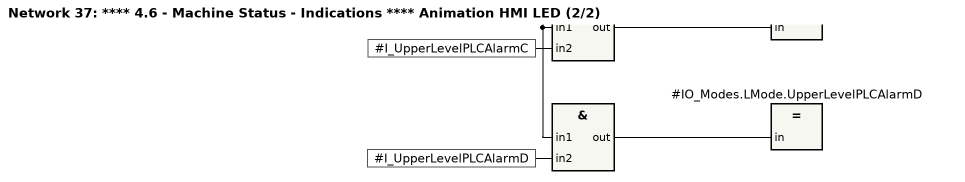
   #IO_Modes.LMode.SafetyOk := "TRUE" AND #I_SafetyOk;
   #IO_Modes.LMode.ZMAlarmABCondition := "TRUE" AND #I_AlarmABCondition;
   #IO_Modes.LMode.ZMAlarmA := "TRUE" AND #I_AlarmA;
   #IO_Modes.LMode.ZMAlarmB := "TRUE" AND #I_AlarmB;
   #IO_Modes.LMode.ZMAlarmC := "TRUE" AND #I_AlarmC;
   #IO_Modes.LMode.ZMAlarmD := "TRUE" AND #I_AlarmD;
   #IO_Modes.LMode.UpperLevelZSAlarmABCondition := "TRUE" AND #I_UpperLevelZSAlarmABCondition;
   #IO_Modes.LMode.UpperLevelZSAlarmA := "TRUE" AND #I_UpperLevelZSAlarmA;
   #IO_Modes.LMode.UpperLevelZSAlarmB := "TRUE" AND #I_UpperLevelZSAlarmB;
   #IO_Modes.LMode.UpperLevelZSAlarmC := "TRUE" AND #I_UpperLevelZSAlarmC;
   #IO_Modes.LMode.UpperLevelZSAlarmD := "TRUE" AND #I_UpperLevelZSAlarmD;
   #IO_Modes.LMode.UpperLevelPLCAlarmABCondition := "TRUE" AND #I_UpperLevelPLCAlarmABCondition;
   #IO_Modes.LMode.UpperLevelPLCAlarmA := "TRUE" AND #I_UpperLevelPLCAlarmA;
   #IO_Modes.LMode.UpperLevelPLCAlarmB := "TRUE" AND #I_UpperLevelPLCAlarmB;
   #IO_Modes.LMode.UpperLevelPLCAlarmC := "TRUE" AND #I_UpperLevelPLCAlarmC;
   #IO_Modes.LMode.UpperLevelPLCAlarmD := "TRUE" AND #I_UpperLevelPLCAlarmD;
END_REGION

REGION Network 38: **** 5.2 - Equations - Flow **** Manual mode is active and the Forced key switch is activated / **** 5.2 - Equations - Flow **** Manual Mode is active and the Forced key switch is activated
   // Manual mode is active and the Forced key switch is activated / Manual Mode is active and the Forced key switch is activated
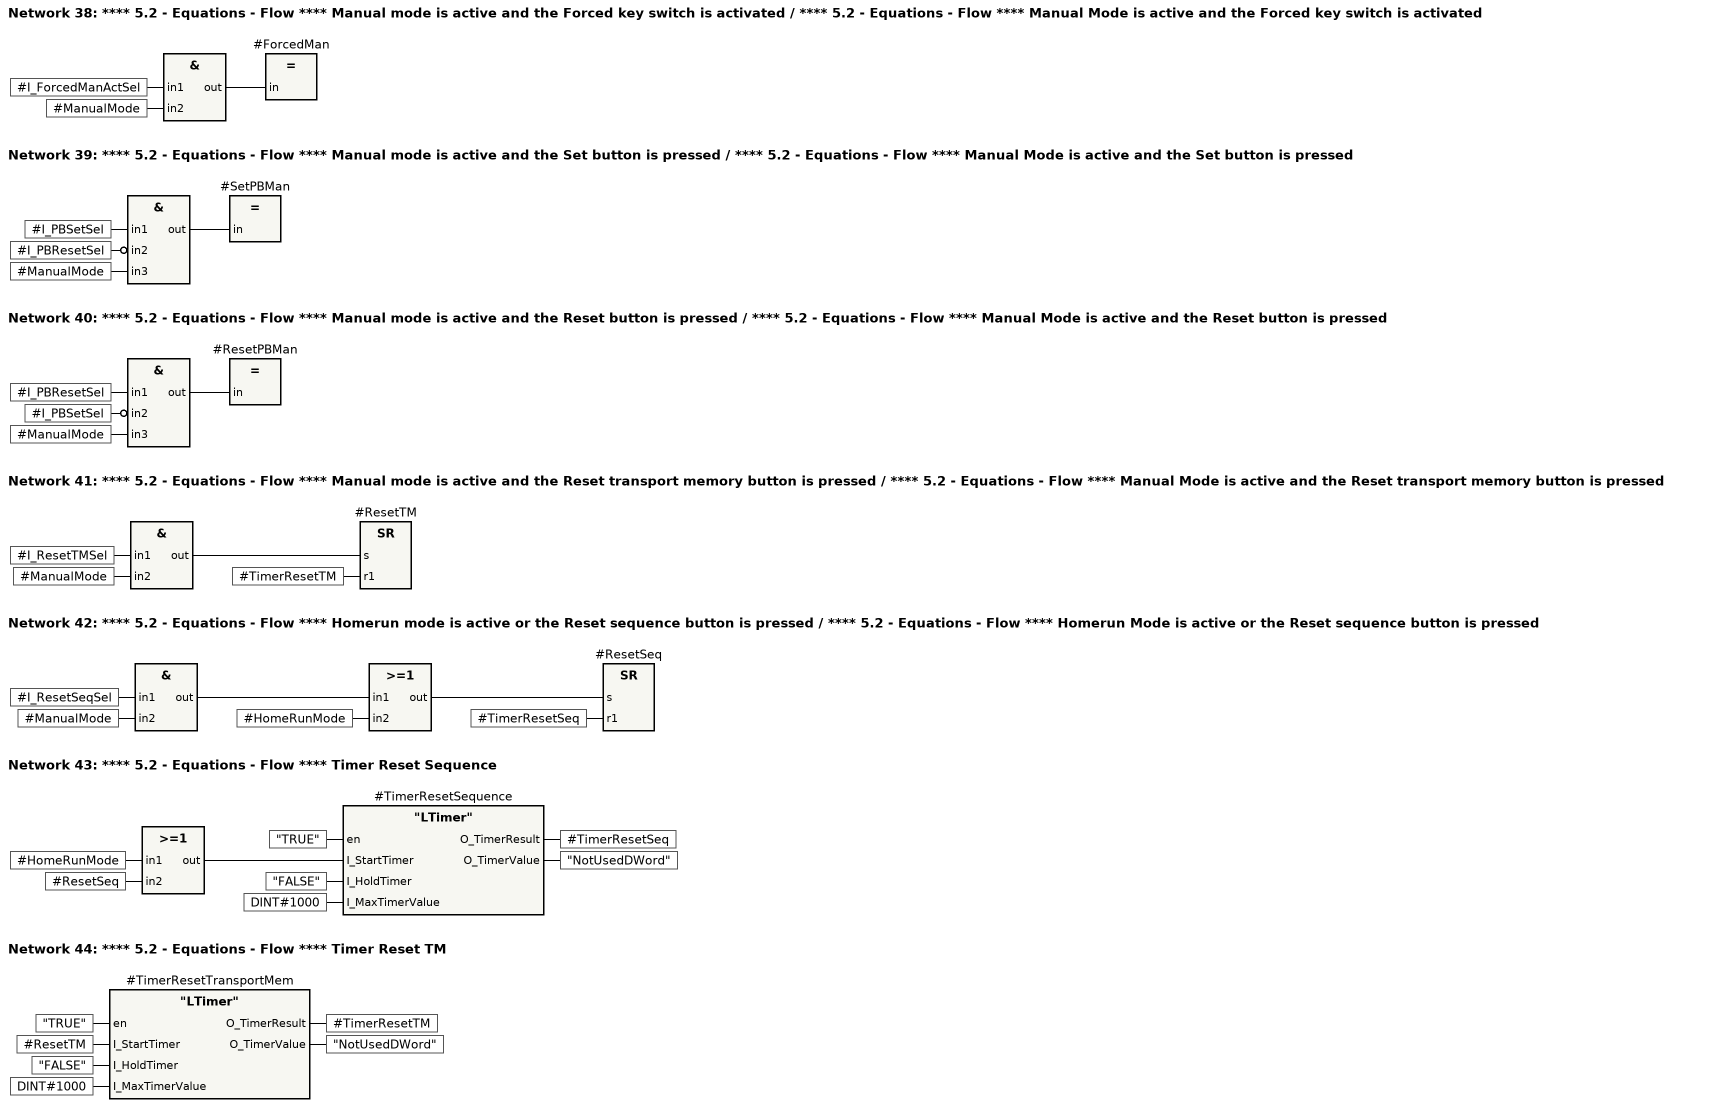
   #ForcedMan := #I_ForcedManActSel AND #ManualMode;
END_REGION

REGION Network 39: **** 5.2 - Equations - Flow **** Manual mode is active and the Set button is pressed / **** 5.2 - Equations - Flow **** Manual Mode is active and the Set button is pressed
   // Manual mode is active and the Set button is pressed / Manual Mode is active and the Set button is pressed
   #SetPBMan := #I_PBSetSel AND NOT #I_PBResetSel AND #ManualMode;
END_REGION

REGION Network 40: **** 5.2 - Equations - Flow **** Manual mode is active and the Reset button is pressed / **** 5.2 - Equations - Flow **** Manual Mode is active and the Reset button is pressed
   // Manual mode is active and the Reset button is pressed / Manual Mode is active and the Reset button is pressed
   #ResetPBMan := #I_PBResetSel AND NOT #I_PBSetSel AND #ManualMode;
END_REGION

REGION Network 41: **** 5.2 - Equations - Flow **** Manual mode is active and the Reset transport memory button is pressed / **** 5.2 - Equations - Flow **** Manual Mode is active and the Reset transport memory button is pressed
   // Manual mode is active and the Reset transport memory button is pressed / Manual Mode is active and the Reset transport memory button is pressed
   IF #I_ResetTMSel AND #ManualMode THEN
       #ResetTM := TRUE;   // SR flip-flop
   END_IF;
   IF #TimerResetTM THEN #ResetTM := FALSE; END_IF;
END_REGION

REGION Network 42: **** 5.2 - Equations - Flow **** Homerun mode is active or the Reset sequence button is pressed / **** 5.2 - Equations - Flow **** Homerun Mode is active or the Reset sequence button is pressed
   // Homerun mode is active or the Reset sequence button is pressed / Homerun Mode is active or the Reset sequence button is pressed
   IF (#I_ResetSeqSel AND #ManualMode) OR #HomeRunMode THEN
       #ResetSeq := TRUE;   // SR flip-flop
   END_IF;
   IF #TimerResetSeq THEN #ResetSeq := FALSE; END_IF;
END_REGION

REGION Network 43: **** 5.2 - Equations - Flow **** Timer Reset Sequence
   // Timer Reset Sequence
   IF "TRUE" THEN
       #TimerResetSequence(I_StartTimer := #HomeRunMode OR #ResetSeq,   // "LTimer"
                           I_HoldTimer := "FALSE",
                           I_MaxTimerValue := DINT#1000,
                           O_TimerResult => #TimerResetSeq,
                           O_TimerValue => "NotUsedDWord");
   END_IF;
END_REGION

REGION Network 44: **** 5.2 - Equations - Flow **** Timer Reset TM
   // Timer Reset TM
   IF "TRUE" THEN
       #TimerResetTransportMem(I_StartTimer := #ResetTM,   // "LTimer"
                               I_HoldTimer := "FALSE",
                               I_MaxTimerValue := DINT#1000,
                               O_TimerResult => #TimerResetTM,
                               O_TimerValue => "NotUsedDWord");
   END_IF;
END_REGION

REGION Network 45: **** 5.2 - Equations - Flow **** Redo after homerun
   // Redo after homerun
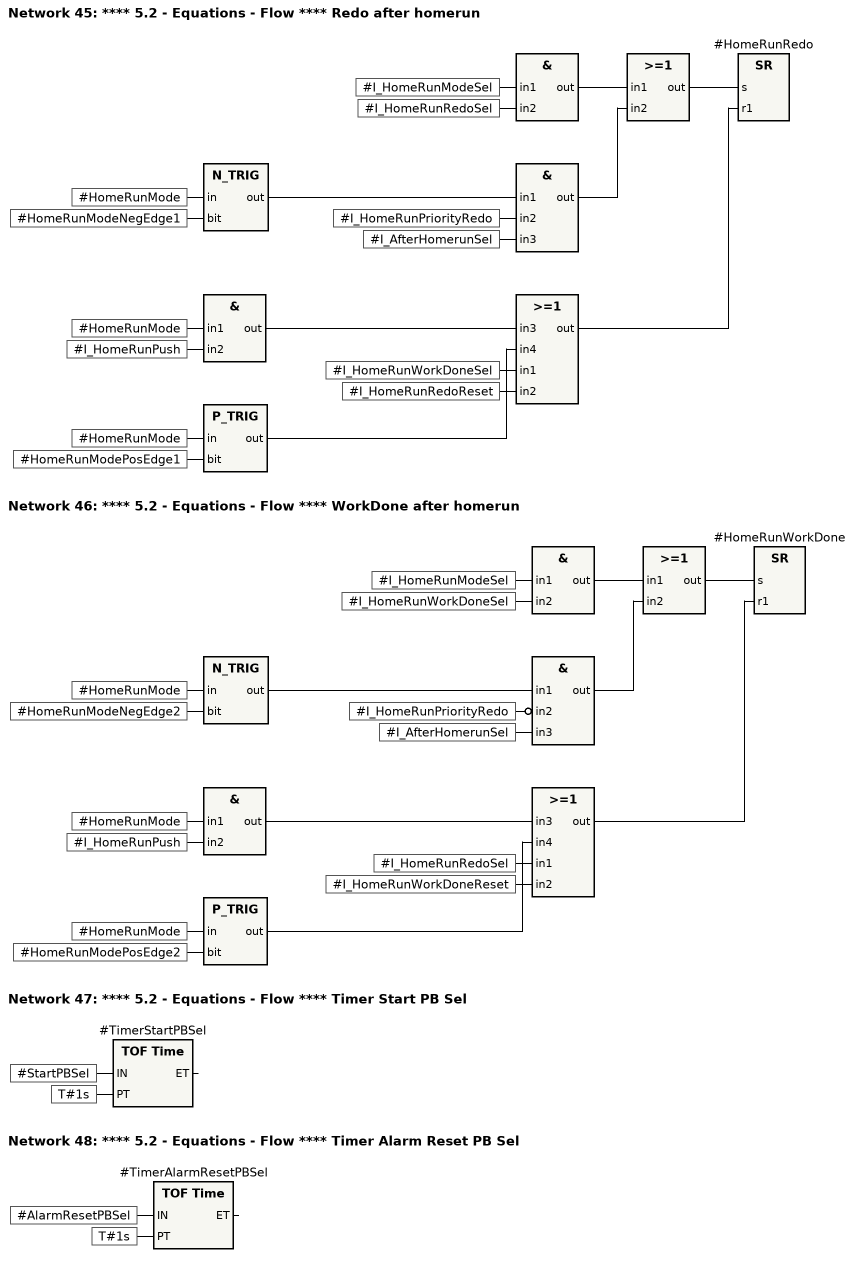
   #_w1 := NOT #HomeRunMode AND #HomeRunModeNegEdge1;   // falling edge
   #HomeRunModeNegEdge1 := #HomeRunMode;
   #_w2 := #HomeRunMode AND NOT #HomeRunModePosEdge1;   // rising edge
   #HomeRunModePosEdge1 := #HomeRunMode;
   IF (#I_HomeRunModeSel AND #I_HomeRunRedoSel) OR (#_w1 AND #I_HomeRunPriorityRedo AND #I_AfterHomerunSel) THEN
       #HomeRunRedo := TRUE;   // SR flip-flop
   END_IF;
   IF (#HomeRunMode AND #I_HomeRunPush) OR #_w2 OR #I_HomeRunWorkDoneSel OR #I_HomeRunRedoReset THEN
       #HomeRunRedo := FALSE;
   END_IF;
END_REGION

REGION Network 46: **** 5.2 - Equations - Flow **** WorkDone after homerun
   // WorkDone after homerun
   #_w1 := NOT #HomeRunMode AND #HomeRunModeNegEdge2;   // falling edge
   #HomeRunModeNegEdge2 := #HomeRunMode;
   #_w2 := #HomeRunMode AND NOT #HomeRunModePosEdge2;   // rising edge
   #HomeRunModePosEdge2 := #HomeRunMode;
   IF (#I_HomeRunModeSel AND #I_HomeRunWorkDoneSel) OR (#_w1 AND NOT #I_HomeRunPriorityRedo AND #I_AfterHomerunSel) THEN
       #HomeRunWorkDone := TRUE;   // SR flip-flop
   END_IF;
   IF (#HomeRunMode AND #I_HomeRunPush) OR #_w2 OR #I_HomeRunRedoSel OR #I_HomeRunWorkDoneReset THEN
       #HomeRunWorkDone := FALSE;
   END_IF;
END_REGION

REGION Network 47: **** 5.2 - Equations - Flow **** Timer Start PB Sel
   // Timer Start PB Sel
   #TimerStartPBSel(IN := #StartPBSel, PT := T#1s);   // TOF
END_REGION

REGION Network 48: **** 5.2 - Equations - Flow **** Timer Alarm Reset PB Sel
   // Timer Alarm Reset PB Sel
   #TimerAlarmResetPBSel(IN := #AlarmResetPBSel, PT := T#1s);   // TOF
END_REGION

REGION Network 49: **** 8 - Outputs **** Set the different bits in the Mode register
   // Set the different bits in the Mode register
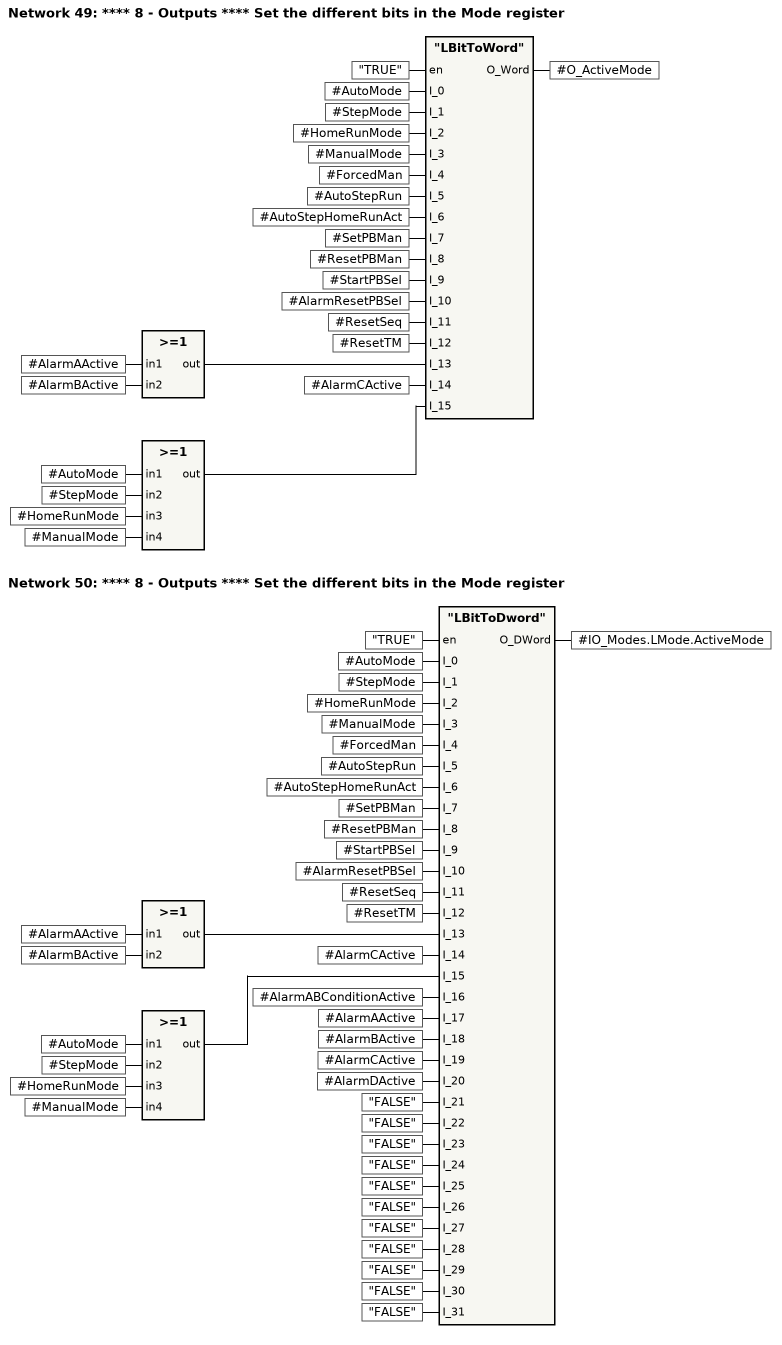
   IF "TRUE" THEN
       "LBitToWord"(I_0 := #AutoMode,
                    I_1 := #StepMode,
                    I_2 := #HomeRunMode,
                    I_3 := #ManualMode,
                    I_4 := #ForcedMan,
                    I_5 := #AutoStepRun,
                    I_6 := #AutoStepHomeRunAct,
                    I_7 := #SetPBMan,
                    I_8 := #ResetPBMan,
                    I_9 := #StartPBSel,
                    I_10 := #AlarmResetPBSel,
                    I_11 := #ResetSeq,
                    I_12 := #ResetTM,
                    I_13 := #AlarmAActive OR #AlarmBActive,
                    I_14 := #AlarmCActive,
                    I_15 := #AutoMode OR #StepMode OR #HomeRunMode OR #ManualMode,
                    O_Word => #O_ActiveMode);
   END_IF;
END_REGION

REGION Network 50: **** 8 - Outputs **** Set the different bits in the Mode register
   // Set the different bits in the Mode register
   IF "TRUE" THEN
       "LBitToDword"(I_0 := #AutoMode,
                     I_1 := #StepMode,
                     I_2 := #HomeRunMode,
                     I_3 := #ManualMode,
                     I_4 := #ForcedMan,
                     I_5 := #AutoStepRun,
                     I_6 := #AutoStepHomeRunAct,
                     I_7 := #SetPBMan,
                     I_8 := #ResetPBMan,
                     I_9 := #StartPBSel,
                     I_10 := #AlarmResetPBSel,
                     I_11 := #ResetSeq,
                     I_12 := #ResetTM,
                     I_13 := #AlarmAActive OR #AlarmBActive,
                     I_14 := #AlarmCActive,
                     I_15 := #AutoMode OR #StepMode OR #HomeRunMode OR #ManualMode,
                     I_16 := #AlarmABConditionActive,
                     I_17 := #AlarmAActive,
                     I_18 := #AlarmBActive,
                     I_19 := #AlarmCActive,
                     I_20 := #AlarmDActive,
                     I_21 := "FALSE",
                     I_22 := "FALSE",
                     I_23 := "FALSE",
                     I_24 := "FALSE",
                     I_25 := "FALSE",
                     I_26 := "FALSE",
                     I_27 := "FALSE",
                     I_28 := "FALSE",
                     I_29 := "FALSE",
                     I_30 := "FALSE",
                     I_31 := "FALSE",
                     O_DWord => #IO_Modes.LMode.ActiveMode);
   END_IF;
END_REGION

REGION Network 51: **** 8 - Outputs **** Set the different bits in the Mode register
   // Set the different bits in the Mode register
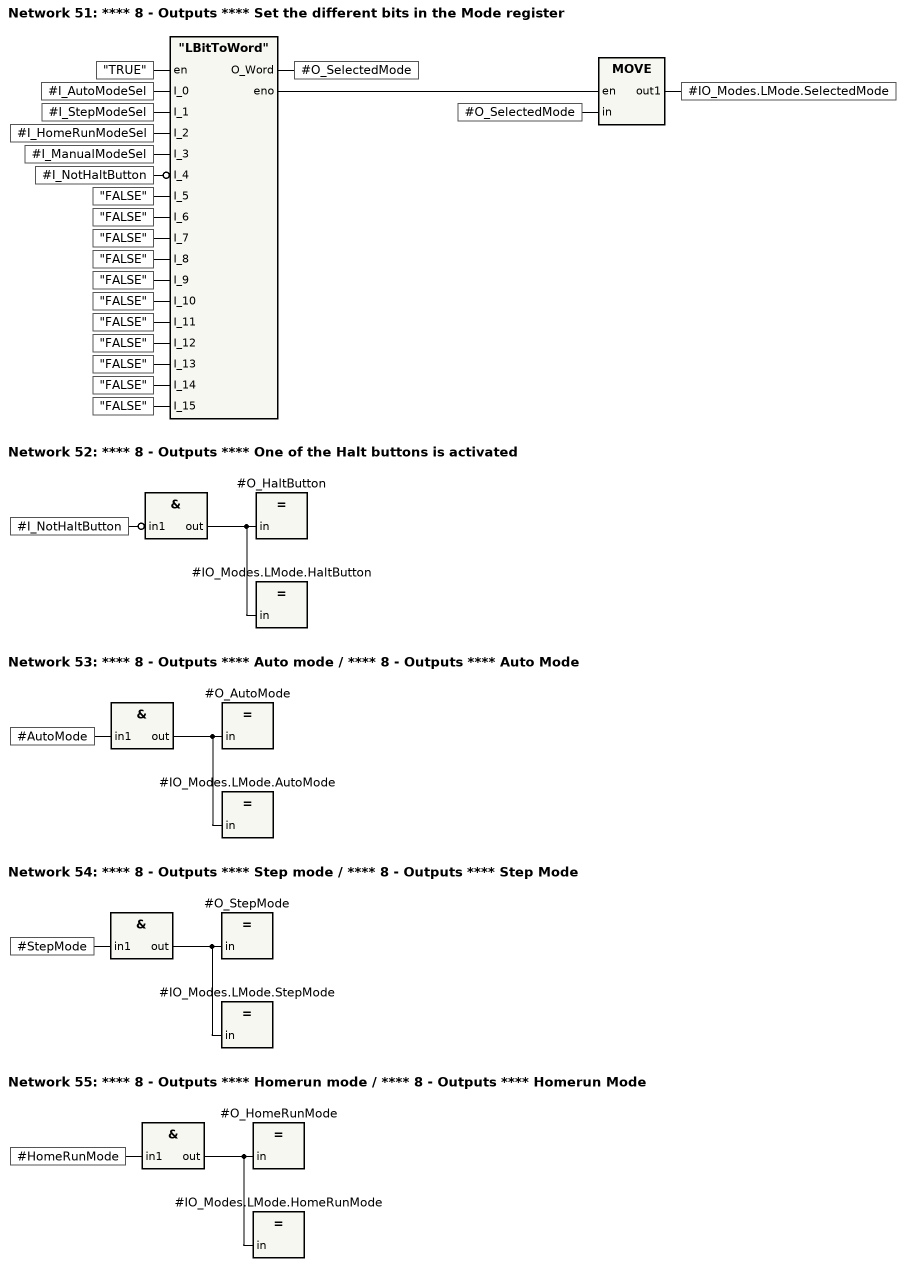
   "LBitToWord"(EN := "TRUE",
                I_0 := #I_AutoModeSel,
                I_1 := #I_StepModeSel,
                I_2 := #I_HomeRunModeSel,
                I_3 := #I_ManualModeSel,
                I_4 := NOT #I_NotHaltButton,
                I_5 := "FALSE",
                I_6 := "FALSE",
                I_7 := "FALSE",
                I_8 := "FALSE",
                I_9 := "FALSE",
                I_10 := "FALSE",
                I_11 := "FALSE",
                I_12 := "FALSE",
                I_13 := "FALSE",
                I_14 := "FALSE",
                I_15 := "FALSE",
                O_Word => #O_SelectedMode,
                ENO => #_w1);
   IF #_w1 THEN #IO_Modes.LMode.SelectedMode := #O_SelectedMode; END_IF;
END_REGION

REGION Network 52: **** 8 - Outputs **** One of the Halt buttons is activated
   // One of the Halt buttons is activated
   #O_HaltButton := NOT #I_NotHaltButton;
   #IO_Modes.LMode.HaltButton := NOT #I_NotHaltButton;
END_REGION

REGION Network 53: **** 8 - Outputs **** Auto mode / **** 8 - Outputs **** Auto Mode
   // Auto mode / Auto Mode
   #O_AutoMode := #AutoMode;
   #IO_Modes.LMode.AutoMode := #AutoMode;
END_REGION

REGION Network 54: **** 8 - Outputs **** Step mode / **** 8 - Outputs **** Step Mode
   // Step mode / Step Mode
   #O_StepMode := #StepMode;
   #IO_Modes.LMode.StepMode := #StepMode;
END_REGION

REGION Network 55: **** 8 - Outputs **** Homerun mode / **** 8 - Outputs **** Homerun Mode
   // Homerun mode / Homerun Mode
   #O_HomeRunMode := #HomeRunMode;
   #IO_Modes.LMode.HomeRunMode := #HomeRunMode;
END_REGION

REGION Network 56: **** 8 - Outputs **** Manual mode / **** 8 - Outputs **** Manual Mode
   // Manual mode / Manual Mode
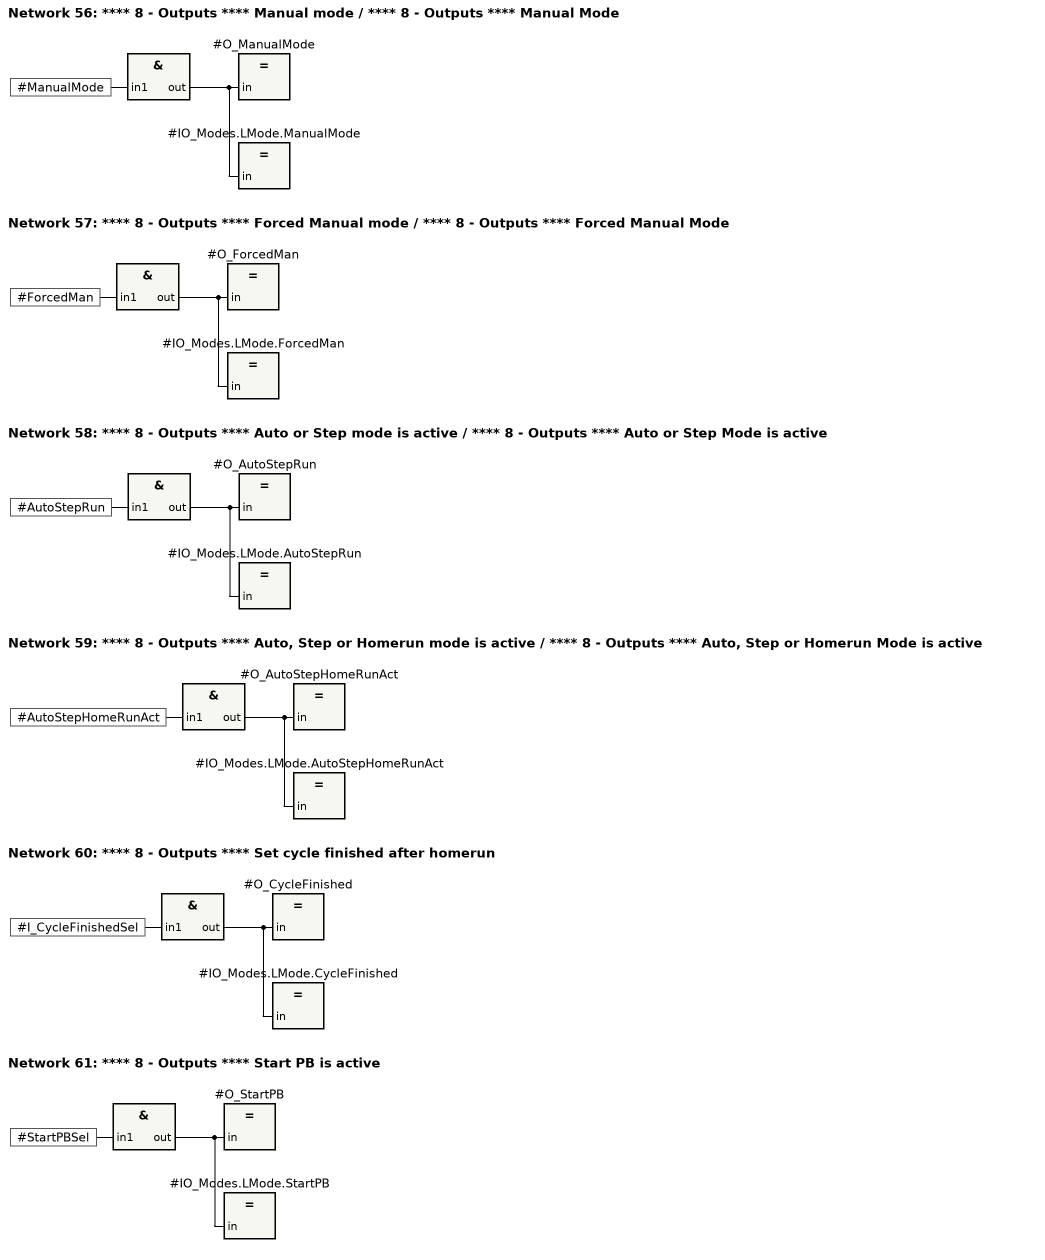
   #O_ManualMode := #ManualMode;
   #IO_Modes.LMode.ManualMode := #ManualMode;
END_REGION

REGION Network 57: **** 8 - Outputs **** Forced Manual mode / **** 8 - Outputs **** Forced Manual Mode
   // Forced Manual mode / Forced Manual Mode
   #O_ForcedMan := #ForcedMan;
   #IO_Modes.LMode.ForcedMan := #ForcedMan;
END_REGION

REGION Network 58: **** 8 - Outputs **** Auto or Step mode is active / **** 8 - Outputs **** Auto or Step Mode is active
   // Auto or Step mode is active / Auto or Step Mode is active
   #O_AutoStepRun := #AutoStepRun;
   #IO_Modes.LMode.AutoStepRun := #AutoStepRun;
END_REGION

REGION Network 59: **** 8 - Outputs **** Auto, Step or Homerun mode is active / **** 8 - Outputs **** Auto, Step or Homerun Mode is active
   // Auto, Step or Homerun mode is active / Auto, Step or Homerun Mode is active
   #O_AutoStepHomeRunAct := #AutoStepHomeRunAct;
   #IO_Modes.LMode.AutoStepHomeRunAct := #AutoStepHomeRunAct;
END_REGION

REGION Network 60: **** 8 - Outputs **** Set cycle finished after homerun
   // Set cycle finished after homerun
   #O_CycleFinished := #I_CycleFinishedSel;
   #IO_Modes.LMode.CycleFinished := #I_CycleFinishedSel;
END_REGION

REGION Network 61: **** 8 - Outputs **** Start PB is active
   // Start PB is active
   #O_StartPB := #StartPBSel;
   #IO_Modes.LMode.StartPB := #StartPBSel;
END_REGION

REGION Network 62: **** 8 - Outputs **** Alarm Reset PB is active
   // Alarm Reset PB is active
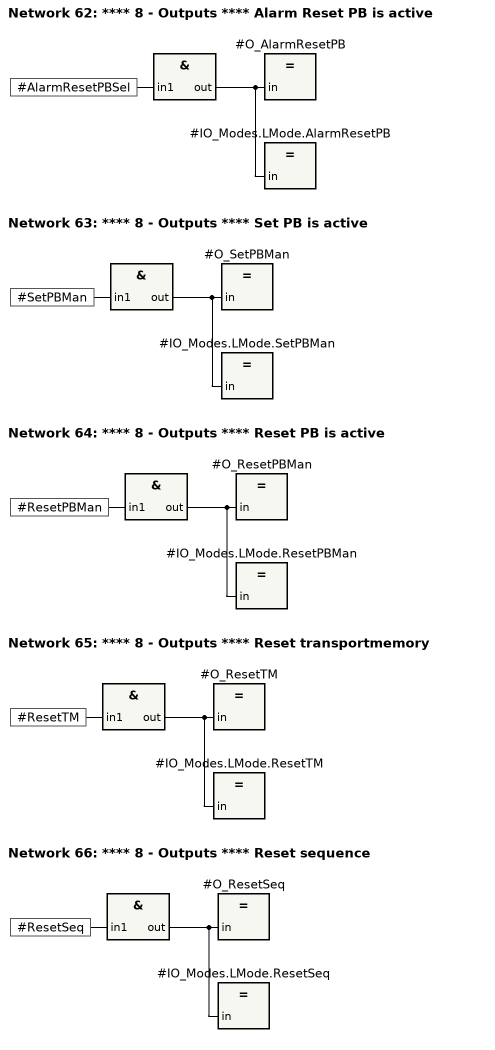
   #O_AlarmResetPB := #AlarmResetPBSel;
   #IO_Modes.LMode.AlarmResetPB := #AlarmResetPBSel;
END_REGION

REGION Network 63: **** 8 - Outputs **** Set PB is active
   // Set PB is active
   #O_SetPBMan := #SetPBMan;
   #IO_Modes.LMode.SetPBMan := #SetPBMan;
END_REGION

REGION Network 64: **** 8 - Outputs **** Reset PB is active
   // Reset PB is active
   #O_ResetPBMan := #ResetPBMan;
   #IO_Modes.LMode.ResetPBMan := #ResetPBMan;
END_REGION

REGION Network 65: **** 8 - Outputs **** Reset transportmemory
   // Reset transportmemory
   #O_ResetTM := #ResetTM;
   #IO_Modes.LMode.ResetTM := #ResetTM;
END_REGION

REGION Network 66: **** 8 - Outputs **** Reset sequence
   // Reset sequence
   #O_ResetSeq := #ResetSeq;
   #IO_Modes.LMode.ResetSeq := #ResetSeq;
END_REGION

REGION Network 67: **** 8 - Outputs **** Auto mode warning / **** 8 - Outputs **** Auto Mode warning
   // Auto mode warning / Auto Mode warning
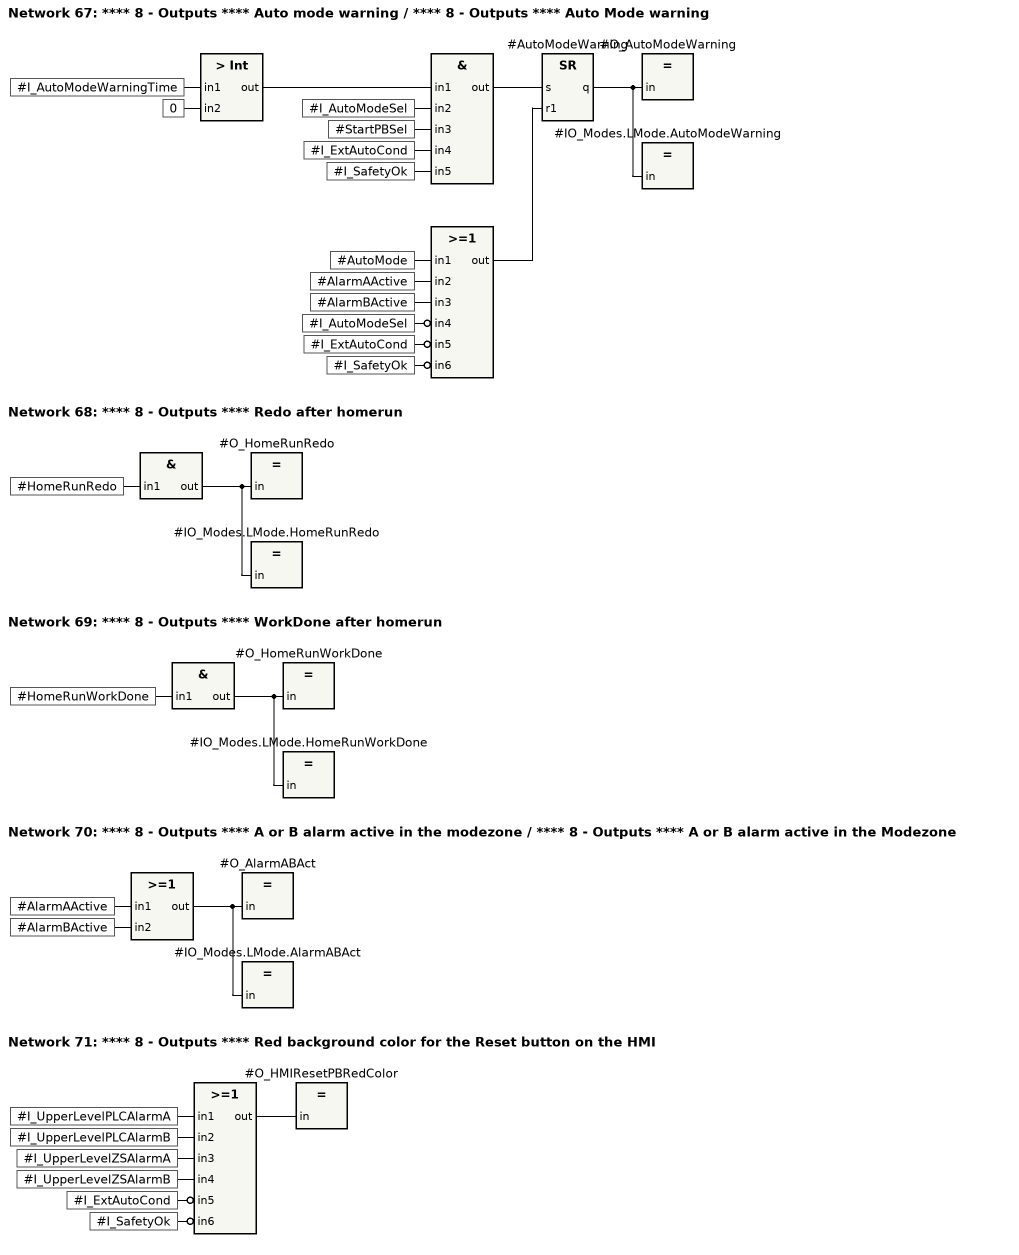
   IF (#I_AutoModeWarningTime > 0) AND #I_AutoModeSel AND #StartPBSel AND #I_ExtAutoCond AND #I_SafetyOk THEN
       #AutoModeWarning := TRUE;   // SR flip-flop
   END_IF;
   IF #AutoMode OR #AlarmAActive OR #AlarmBActive OR NOT #I_AutoModeSel OR NOT #I_ExtAutoCond OR NOT #I_SafetyOk THEN
       #AutoModeWarning := FALSE;
   END_IF;
   #O_AutoModeWarning := #AutoModeWarning;
   #IO_Modes.LMode.AutoModeWarning := #AutoModeWarning;
END_REGION

REGION Network 68: **** 8 - Outputs **** Redo after homerun
   // Redo after homerun
   #O_HomeRunRedo := #HomeRunRedo;
   #IO_Modes.LMode.HomeRunRedo := #HomeRunRedo;
END_REGION

REGION Network 69: **** 8 - Outputs **** WorkDone after homerun
   // WorkDone after homerun
   #O_HomeRunWorkDone := #HomeRunWorkDone;
   #IO_Modes.LMode.HomeRunWorkDone := #HomeRunWorkDone;
END_REGION

REGION Network 70: **** 8 - Outputs **** A or B alarm active in the modezone / **** 8 - Outputs **** A or B alarm active in the Modezone
   // A or B alarm active in the modezone / A or B alarm active in the Modezone
   #O_AlarmABAct := #AlarmAActive OR #AlarmBActive;
   #IO_Modes.LMode.AlarmABAct := #O_AlarmABAct;
END_REGION

REGION Network 71: **** 8 - Outputs **** Red background color for the Reset button on the HMI
   #O_HMIResetPBRedColor := #I_UpperLevelPLCAlarmA OR #I_UpperLevelPLCAlarmB OR #I_UpperLevelZSAlarmA OR #I_UpperLevelZSAlarmB OR NOT #I_ExtAutoCond OR NOT #I_SafetyOk;
END_REGION

REGION Network 72: **** 8 - Outputs **** Alarm AB condition
   // Alarm AB condition
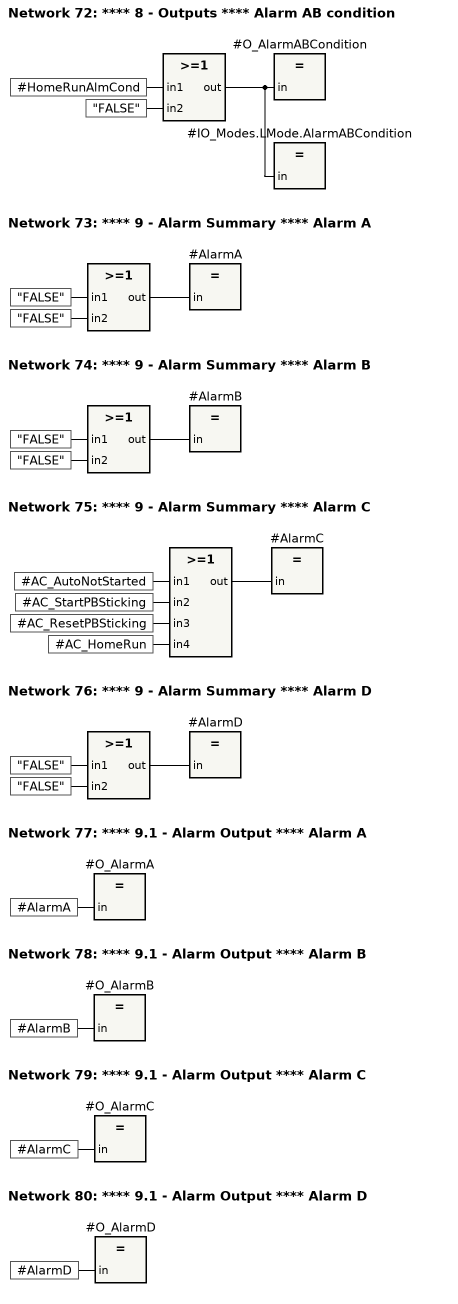
   #O_AlarmABCondition := #HomeRunAlmCond OR "FALSE";
   #IO_Modes.LMode.AlarmABCondition := #O_AlarmABCondition;
END_REGION

REGION Network 73: **** 9 - Alarm Summary **** Alarm A
   // Summary of alarms A
   #AlarmA := "FALSE" OR "FALSE";
END_REGION

REGION Network 74: **** 9 - Alarm Summary **** Alarm B
   // Summary of alarms B
   #AlarmB := "FALSE" OR "FALSE";
END_REGION

REGION Network 75: **** 9 - Alarm Summary **** Alarm C
   // Summary of alarms C
   #AlarmC := #AC_AutoNotStarted OR #AC_StartPBSticking OR #AC_ResetPBSticking OR #AC_HomeRun;
END_REGION

REGION Network 76: **** 9 - Alarm Summary **** Alarm D
   // Summary of alarms D
   #AlarmD := "FALSE" OR "FALSE";
END_REGION

REGION Network 77: **** 9.1 - Alarm Output **** Alarm A
   // Summary of alarms A
   #O_AlarmA := #AlarmA;
END_REGION

REGION Network 78: **** 9.1 - Alarm Output **** Alarm B
   // Summary of alarms B
   #O_AlarmB := #AlarmB;
END_REGION

REGION Network 79: **** 9.1 - Alarm Output **** Alarm C
   // Summary of alarms C
   #O_AlarmC := #AlarmC;
END_REGION

REGION Network 80: **** 9.1 - Alarm Output **** Alarm D
   // Summary of alarms D
   #O_AlarmD := #AlarmD;
END_REGION

REGION Network 81: **** 9.2 - Alarm DWord**** Alarm To DWord
   // Alarm Word
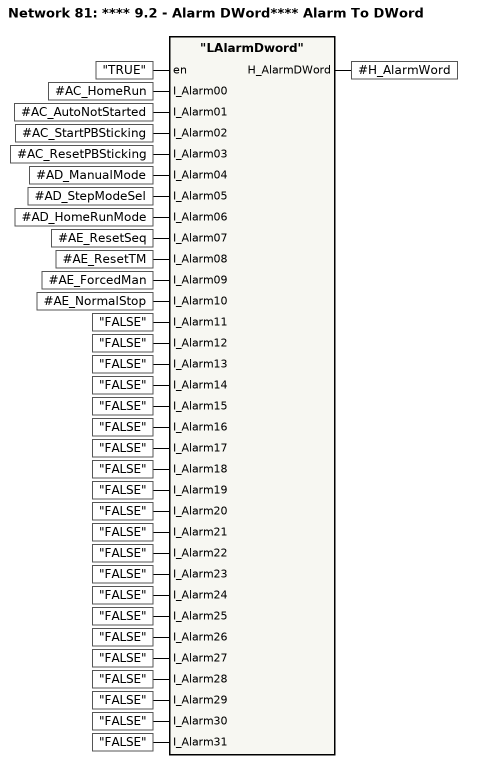
   IF "TRUE" THEN
       "LAlarmDword"(I_Alarm00 := #AC_HomeRun,
                     I_Alarm01 := #AC_AutoNotStarted,
                     I_Alarm02 := #AC_StartPBSticking,
                     I_Alarm03 := #AC_ResetPBSticking,
                     I_Alarm04 := #AD_ManualMode,
                     I_Alarm05 := #AD_StepModeSel,
                     I_Alarm06 := #AD_HomeRunMode,
                     I_Alarm07 := #AE_ResetSeq,
                     I_Alarm08 := #AE_ResetTM,
                     I_Alarm09 := #AE_ForcedMan,
                     I_Alarm10 := #AE_NormalStop,
                     I_Alarm11 := "FALSE",
                     I_Alarm12 := "FALSE",
                     I_Alarm13 := "FALSE",
                     I_Alarm14 := "FALSE",
                     I_Alarm15 := "FALSE",
                     I_Alarm16 := "FALSE",
                     I_Alarm17 := "FALSE",
                     I_Alarm18 := "FALSE",
                     I_Alarm19 := "FALSE",
                     I_Alarm20 := "FALSE",
                     I_Alarm21 := "FALSE",
                     I_Alarm22 := "FALSE",
                     I_Alarm23 := "FALSE",
                     I_Alarm24 := "FALSE",
                     I_Alarm25 := "FALSE",
                     I_Alarm26 := "FALSE",
                     I_Alarm27 := "FALSE",
                     I_Alarm28 := "FALSE",
                     I_Alarm29 := "FALSE",
                     I_Alarm30 := "FALSE",
                     I_Alarm31 := "FALSE",
                     H_AlarmDWord => #H_AlarmWord);
   END_IF;
END_REGION
END_FUNCTION_BLOCK
